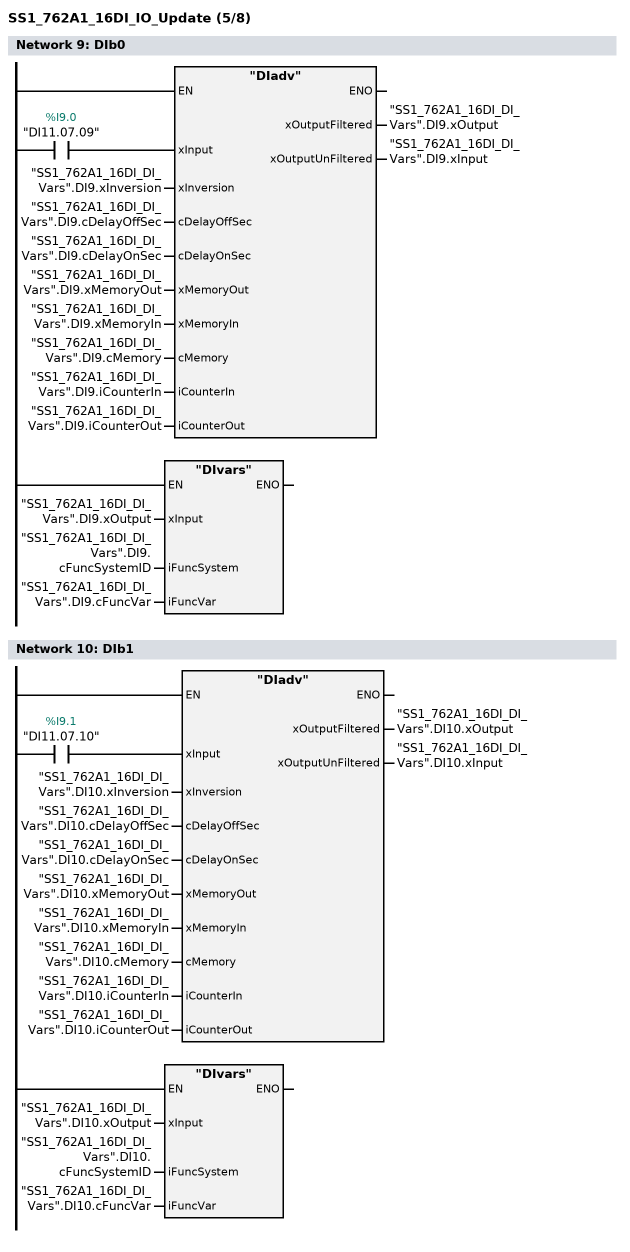
   RUNG wire#powerrail
      "DIadv"(xInput := wire#w1, xInversion := "SS1_762A1_16DI_DI_Vars".DI9.xInversion, cDelayOffSec := "SS1_762A1_16DI_DI_Vars".DI9.cDelayOffSec, cDelayOnSec := "SS1_762A1_16DI_DI_Vars".DI9.cDelayOnSec, xMemoryOut := "SS1_762A1_16DI_DI_Vars".DI9.xMemoryOut, xMemoryIn := "SS1_762A1_16DI_DI_Vars".DI9.xMemoryIn, cMemory := "SS1_762A1_16DI_DI_Vars".DI9.cMemory, iCounterIn := "SS1_762A1_16DI_DI_Vars".DI9.iCounterIn, iCounterOut := "SS1_762A1_16DI_DI_Vars".DI9.iCounterOut, xOutputFiltered => "SS1_762A1_16DI_DI_Vars".DI9.xOutput, xOutputUnFiltered => "SS1_762A1_16DI_DI_Vars".DI9.xInput)
   END_RUNG
   RUNG wire#powerrail
      Contact( "DI11.07.09" )
   END_RUNG wire#w1
   RUNG wire#powerrail
      "DIvars"(xInput := "SS1_762A1_16DI_DI_Vars".DI9.xOutput, iFuncSystem := "SS1_762A1_16DI_DI_Vars".DI9.cFuncSystemID, iFuncVar := "SS1_762A1_16DI_DI_Vars".DI9.cFuncVar)
   END_RUNG
   // the same network as SCL:
   "DIadv"(xInput := "DI11.07.09",
           xInversion := "SS1_762A1_16DI_DI_Vars".DI9.xInversion,
           cDelayOffSec := "SS1_762A1_16DI_DI_Vars".DI9.cDelayOffSec,
           cDelayOnSec := "SS1_762A1_16DI_DI_Vars".DI9.cDelayOnSec,
           xMemoryOut := "SS1_762A1_16DI_DI_Vars".DI9.xMemoryOut,
           xMemoryIn := "SS1_762A1_16DI_DI_Vars".DI9.xMemoryIn,
           cMemory := "SS1_762A1_16DI_DI_Vars".DI9.cMemory,
           iCounterIn := "SS1_762A1_16DI_DI_Vars".DI9.iCounterIn,
           iCounterOut := "SS1_762A1_16DI_DI_Vars".DI9.iCounterOut,
           xOutputFiltered => "SS1_762A1_16DI_DI_Vars".DI9.xOutput,
           xOutputUnFiltered => "SS1_762A1_16DI_DI_Vars".DI9.xInput);
   "DIvars"(xInput := "SS1_762A1_16DI_DI_Vars".DI9.xOutput,
            iFuncSystem := "SS1_762A1_16DI_DI_Vars".DI9.cFuncSystemID,
            iFuncVar := "SS1_762A1_16DI_DI_Vars".DI9.cFuncVar);
END_REGION

REGION Network 10: DIb1
   RUNG wire#powerrail
      "DIadv"(xInput := wire#w1, xInversion := "SS1_762A1_16DI_DI_Vars".DI10.xInversion, cDelayOffSec := "SS1_762A1_16DI_DI_Vars".DI10.cDelayOffSec, cDelayOnSec := "SS1_762A1_16DI_DI_Vars".DI10.cDelayOnSec, xMemoryOut := "SS1_762A1_16DI_DI_Vars".DI10.xMemoryOut, xMemoryIn := "SS1_762A1_16DI_DI_Vars".DI10.xMemoryIn, cMemory := "SS1_762A1_16DI_DI_Vars".DI10.cMemory, iCounterIn := "SS1_762A1_16DI_DI_Vars".DI10.iCounterIn, iCounterOut := "SS1_762A1_16DI_DI_Vars".DI10.iCounterOut, xOutputFiltered => "SS1_762A1_16DI_DI_Vars".DI10.xOutput, xOutputUnFiltered => "SS1_762A1_16DI_DI_Vars".DI10.xInput)
   END_RUNG
   RUNG wire#powerrail
      Contact( "DI11.07.10" )
   END_RUNG wire#w1
   RUNG wire#powerrail
      "DIvars"(xInput := "SS1_762A1_16DI_DI_Vars".DI10.xOutput, iFuncSystem := "SS1_762A1_16DI_DI_Vars".DI10.cFuncSystemID, iFuncVar := "SS1_762A1_16DI_DI_Vars".DI10.cFuncVar)
   END_RUNG
   // the same network as SCL:
   "DIadv"(xInput := "DI11.07.10",
           xInversion := "SS1_762A1_16DI_DI_Vars".DI10.xInversion,
           cDelayOffSec := "SS1_762A1_16DI_DI_Vars".DI10.cDelayOffSec,
           cDelayOnSec := "SS1_762A1_16DI_DI_Vars".DI10.cDelayOnSec,
           xMemoryOut := "SS1_762A1_16DI_DI_Vars".DI10.xMemoryOut,
           xMemoryIn := "SS1_762A1_16DI_DI_Vars".DI10.xMemoryIn,
           cMemory := "SS1_762A1_16DI_DI_Vars".DI10.cMemory,
           iCounterIn := "SS1_762A1_16DI_DI_Vars".DI10.iCounterIn,
           iCounterOut := "SS1_762A1_16DI_DI_Vars".DI10.iCounterOut,
           xOutputFiltered => "SS1_762A1_16DI_DI_Vars".DI10.xOutput,
           xOutputUnFiltered => "SS1_762A1_16DI_DI_Vars".DI10.xInput);
   "DIvars"(xInput := "SS1_762A1_16DI_DI_Vars".DI10.xOutput,
            iFuncSystem := "SS1_762A1_16DI_DI_Vars".DI10.cFuncSystemID,
            iFuncVar := "SS1_762A1_16DI_DI_Vars".DI10.cFuncVar);
END_REGION

REGION Network 11: DIb2
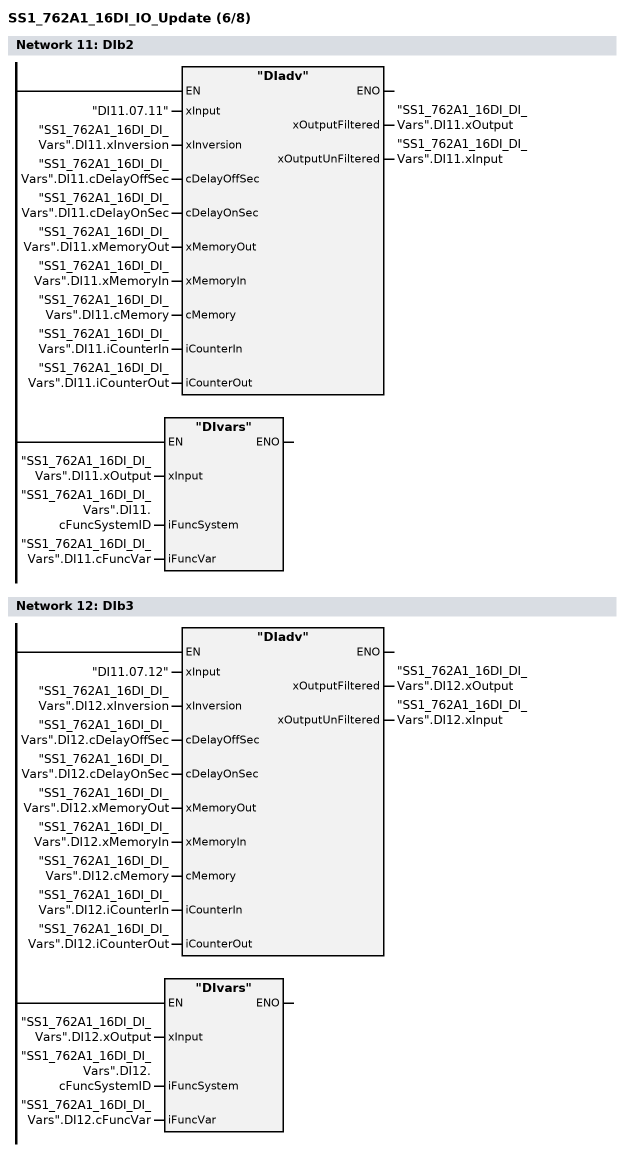
   RUNG wire#powerrail
      "DIadv"(xInput := "DI11.07.11", xInversion := "SS1_762A1_16DI_DI_Vars".DI11.xInversion, cDelayOffSec := "SS1_762A1_16DI_DI_Vars".DI11.cDelayOffSec, cDelayOnSec := "SS1_762A1_16DI_DI_Vars".DI11.cDelayOnSec, xMemoryOut := "SS1_762A1_16DI_DI_Vars".DI11.xMemoryOut, xMemoryIn := "SS1_762A1_16DI_DI_Vars".DI11.xMemoryIn, cMemory := "SS1_762A1_16DI_DI_Vars".DI11.cMemory, iCounterIn := "SS1_762A1_16DI_DI_Vars".DI11.iCounterIn, iCounterOut := "SS1_762A1_16DI_DI_Vars".DI11.iCounterOut, xOutputFiltered => "SS1_762A1_16DI_DI_Vars".DI11.xOutput, xOutputUnFiltered => "SS1_762A1_16DI_DI_Vars".DI11.xInput)
   END_RUNG
   RUNG wire#powerrail
      "DIvars"(xInput := "SS1_762A1_16DI_DI_Vars".DI11.xOutput, iFuncSystem := "SS1_762A1_16DI_DI_Vars".DI11.cFuncSystemID, iFuncVar := "SS1_762A1_16DI_DI_Vars".DI11.cFuncVar)
   END_RUNG
   // the same network as SCL:
   "DIadv"(xInput := "DI11.07.11",
           xInversion := "SS1_762A1_16DI_DI_Vars".DI11.xInversion,
           cDelayOffSec := "SS1_762A1_16DI_DI_Vars".DI11.cDelayOffSec,
           cDelayOnSec := "SS1_762A1_16DI_DI_Vars".DI11.cDelayOnSec,
           xMemoryOut := "SS1_762A1_16DI_DI_Vars".DI11.xMemoryOut,
           xMemoryIn := "SS1_762A1_16DI_DI_Vars".DI11.xMemoryIn,
           cMemory := "SS1_762A1_16DI_DI_Vars".DI11.cMemory,
           iCounterIn := "SS1_762A1_16DI_DI_Vars".DI11.iCounterIn,
           iCounterOut := "SS1_762A1_16DI_DI_Vars".DI11.iCounterOut,
           xOutputFiltered => "SS1_762A1_16DI_DI_Vars".DI11.xOutput,
           xOutputUnFiltered => "SS1_762A1_16DI_DI_Vars".DI11.xInput);
   "DIvars"(xInput := "SS1_762A1_16DI_DI_Vars".DI11.xOutput,
            iFuncSystem := "SS1_762A1_16DI_DI_Vars".DI11.cFuncSystemID,
            iFuncVar := "SS1_762A1_16DI_DI_Vars".DI11.cFuncVar);
END_REGION

REGION Network 12: DIb3
   RUNG wire#powerrail
      "DIadv"(xInput := "DI11.07.12", xInversion := "SS1_762A1_16DI_DI_Vars".DI12.xInversion, cDelayOffSec := "SS1_762A1_16DI_DI_Vars".DI12.cDelayOffSec, cDelayOnSec := "SS1_762A1_16DI_DI_Vars".DI12.cDelayOnSec, xMemoryOut := "SS1_762A1_16DI_DI_Vars".DI12.xMemoryOut, xMemoryIn := "SS1_762A1_16DI_DI_Vars".DI12.xMemoryIn, cMemory := "SS1_762A1_16DI_DI_Vars".DI12.cMemory, iCounterIn := "SS1_762A1_16DI_DI_Vars".DI12.iCounterIn, iCounterOut := "SS1_762A1_16DI_DI_Vars".DI12.iCounterOut, xOutputFiltered => "SS1_762A1_16DI_DI_Vars".DI12.xOutput, xOutputUnFiltered => "SS1_762A1_16DI_DI_Vars".DI12.xInput)
   END_RUNG
   RUNG wire#powerrail
      "DIvars"(xInput := "SS1_762A1_16DI_DI_Vars".DI12.xOutput, iFuncSystem := "SS1_762A1_16DI_DI_Vars".DI12.cFuncSystemID, iFuncVar := "SS1_762A1_16DI_DI_Vars".DI12.cFuncVar)
   END_RUNG
   // the same network as SCL:
   "DIadv"(xInput := "DI11.07.12",
           xInversion := "SS1_762A1_16DI_DI_Vars".DI12.xInversion,
           cDelayOffSec := "SS1_762A1_16DI_DI_Vars".DI12.cDelayOffSec,
           cDelayOnSec := "SS1_762A1_16DI_DI_Vars".DI12.cDelayOnSec,
           xMemoryOut := "SS1_762A1_16DI_DI_Vars".DI12.xMemoryOut,
           xMemoryIn := "SS1_762A1_16DI_DI_Vars".DI12.xMemoryIn,
           cMemory := "SS1_762A1_16DI_DI_Vars".DI12.cMemory,
           iCounterIn := "SS1_762A1_16DI_DI_Vars".DI12.iCounterIn,
           iCounterOut := "SS1_762A1_16DI_DI_Vars".DI12.iCounterOut,
           xOutputFiltered => "SS1_762A1_16DI_DI_Vars".DI12.xOutput,
           xOutputUnFiltered => "SS1_762A1_16DI_DI_Vars".DI12.xInput);
   "DIvars"(xInput := "SS1_762A1_16DI_DI_Vars".DI12.xOutput,
            iFuncSystem := "SS1_762A1_16DI_DI_Vars".DI12.cFuncSystemID,
            iFuncVar := "SS1_762A1_16DI_DI_Vars".DI12.cFuncVar);
END_REGION

REGION Network 13: DIb4
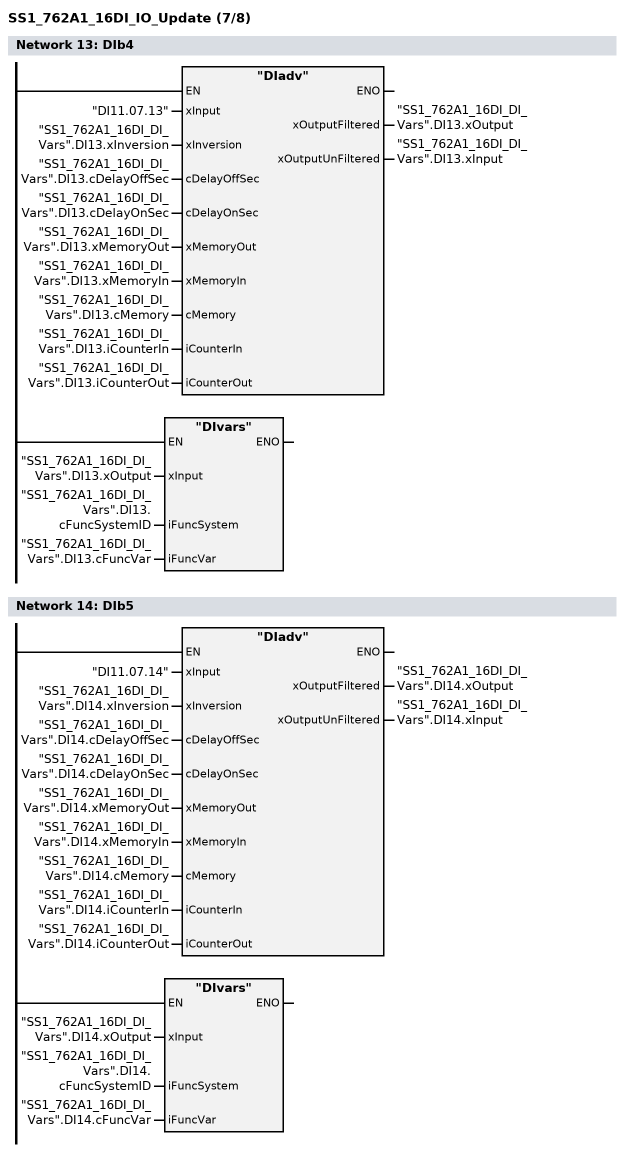
   RUNG wire#powerrail
      "DIadv"(xInput := "DI11.07.13", xInversion := "SS1_762A1_16DI_DI_Vars".DI13.xInversion, cDelayOffSec := "SS1_762A1_16DI_DI_Vars".DI13.cDelayOffSec, cDelayOnSec := "SS1_762A1_16DI_DI_Vars".DI13.cDelayOnSec, xMemoryOut := "SS1_762A1_16DI_DI_Vars".DI13.xMemoryOut, xMemoryIn := "SS1_762A1_16DI_DI_Vars".DI13.xMemoryIn, cMemory := "SS1_762A1_16DI_DI_Vars".DI13.cMemory, iCounterIn := "SS1_762A1_16DI_DI_Vars".DI13.iCounterIn, iCounterOut := "SS1_762A1_16DI_DI_Vars".DI13.iCounterOut, xOutputFiltered => "SS1_762A1_16DI_DI_Vars".DI13.xOutput, xOutputUnFiltered => "SS1_762A1_16DI_DI_Vars".DI13.xInput)
   END_RUNG
   RUNG wire#powerrail
      "DIvars"(xInput := "SS1_762A1_16DI_DI_Vars".DI13.xOutput, iFuncSystem := "SS1_762A1_16DI_DI_Vars".DI13.cFuncSystemID, iFuncVar := "SS1_762A1_16DI_DI_Vars".DI13.cFuncVar)
   END_RUNG
   // the same network as SCL:
   "DIadv"(xInput := "DI11.07.13",
           xInversion := "SS1_762A1_16DI_DI_Vars".DI13.xInversion,
           cDelayOffSec := "SS1_762A1_16DI_DI_Vars".DI13.cDelayOffSec,
           cDelayOnSec := "SS1_762A1_16DI_DI_Vars".DI13.cDelayOnSec,
           xMemoryOut := "SS1_762A1_16DI_DI_Vars".DI13.xMemoryOut,
           xMemoryIn := "SS1_762A1_16DI_DI_Vars".DI13.xMemoryIn,
           cMemory := "SS1_762A1_16DI_DI_Vars".DI13.cMemory,
           iCounterIn := "SS1_762A1_16DI_DI_Vars".DI13.iCounterIn,
           iCounterOut := "SS1_762A1_16DI_DI_Vars".DI13.iCounterOut,
           xOutputFiltered => "SS1_762A1_16DI_DI_Vars".DI13.xOutput,
           xOutputUnFiltered => "SS1_762A1_16DI_DI_Vars".DI13.xInput);
   "DIvars"(xInput := "SS1_762A1_16DI_DI_Vars".DI13.xOutput,
            iFuncSystem := "SS1_762A1_16DI_DI_Vars".DI13.cFuncSystemID,
            iFuncVar := "SS1_762A1_16DI_DI_Vars".DI13.cFuncVar);
END_REGION

REGION Network 14: DIb5
   RUNG wire#powerrail
      "DIadv"(xInput := "DI11.07.14", xInversion := "SS1_762A1_16DI_DI_Vars".DI14.xInversion, cDelayOffSec := "SS1_762A1_16DI_DI_Vars".DI14.cDelayOffSec, cDelayOnSec := "SS1_762A1_16DI_DI_Vars".DI14.cDelayOnSec, xMemoryOut := "SS1_762A1_16DI_DI_Vars".DI14.xMemoryOut, xMemoryIn := "SS1_762A1_16DI_DI_Vars".DI14.xMemoryIn, cMemory := "SS1_762A1_16DI_DI_Vars".DI14.cMemory, iCounterIn := "SS1_762A1_16DI_DI_Vars".DI14.iCounterIn, iCounterOut := "SS1_762A1_16DI_DI_Vars".DI14.iCounterOut, xOutputFiltered => "SS1_762A1_16DI_DI_Vars".DI14.xOutput, xOutputUnFiltered => "SS1_762A1_16DI_DI_Vars".DI14.xInput)
   END_RUNG
   RUNG wire#powerrail
      "DIvars"(xInput := "SS1_762A1_16DI_DI_Vars".DI14.xOutput, iFuncSystem := "SS1_762A1_16DI_DI_Vars".DI14.cFuncSystemID, iFuncVar := "SS1_762A1_16DI_DI_Vars".DI14.cFuncVar)
   END_RUNG
   // the same network as SCL:
   "DIadv"(xInput := "DI11.07.14",
           xInversion := "SS1_762A1_16DI_DI_Vars".DI14.xInversion,
           cDelayOffSec := "SS1_762A1_16DI_DI_Vars".DI14.cDelayOffSec,
           cDelayOnSec := "SS1_762A1_16DI_DI_Vars".DI14.cDelayOnSec,
           xMemoryOut := "SS1_762A1_16DI_DI_Vars".DI14.xMemoryOut,
           xMemoryIn := "SS1_762A1_16DI_DI_Vars".DI14.xMemoryIn,
           cMemory := "SS1_762A1_16DI_DI_Vars".DI14.cMemory,
           iCounterIn := "SS1_762A1_16DI_DI_Vars".DI14.iCounterIn,
           iCounterOut := "SS1_762A1_16DI_DI_Vars".DI14.iCounterOut,
           xOutputFiltered => "SS1_762A1_16DI_DI_Vars".DI14.xOutput,
           xOutputUnFiltered => "SS1_762A1_16DI_DI_Vars".DI14.xInput);
   "DIvars"(xInput := "SS1_762A1_16DI_DI_Vars".DI14.xOutput,
            iFuncSystem := "SS1_762A1_16DI_DI_Vars".DI14.cFuncSystemID,
            iFuncVar := "SS1_762A1_16DI_DI_Vars".DI14.cFuncVar);
END_REGION

REGION Network 15: DIb6
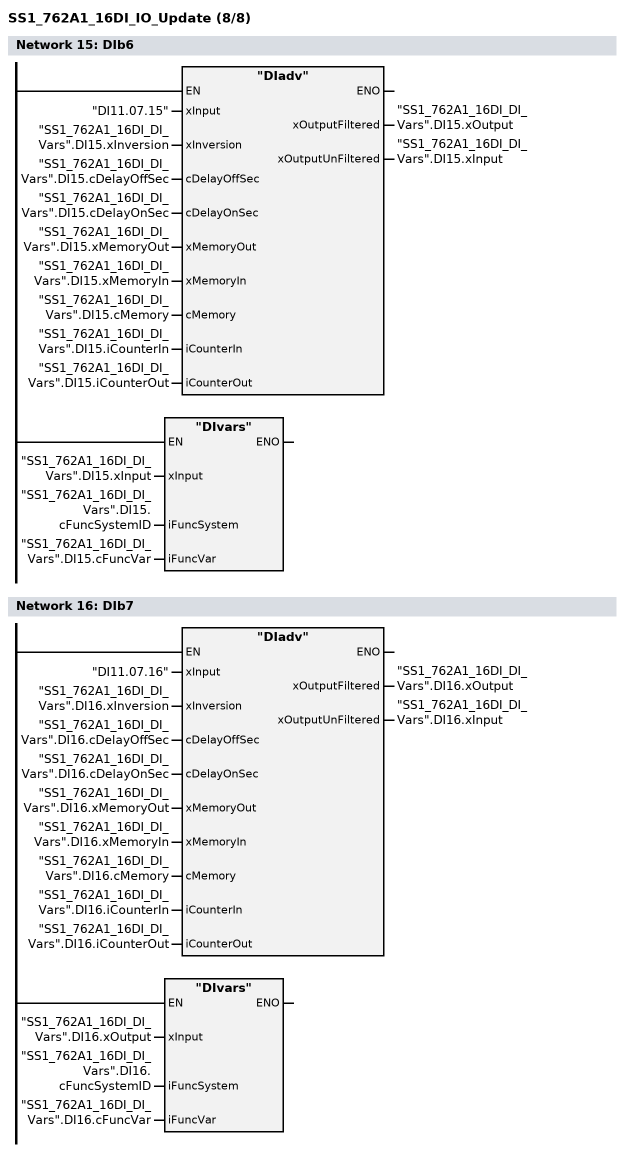
   RUNG wire#powerrail
      "DIadv"(xInput := "DI11.07.15", xInversion := "SS1_762A1_16DI_DI_Vars".DI15.xInversion, cDelayOffSec := "SS1_762A1_16DI_DI_Vars".DI15.cDelayOffSec, cDelayOnSec := "SS1_762A1_16DI_DI_Vars".DI15.cDelayOnSec, xMemoryOut := "SS1_762A1_16DI_DI_Vars".DI15.xMemoryOut, xMemoryIn := "SS1_762A1_16DI_DI_Vars".DI15.xMemoryIn, cMemory := "SS1_762A1_16DI_DI_Vars".DI15.cMemory, iCounterIn := "SS1_762A1_16DI_DI_Vars".DI15.iCounterIn, iCounterOut := "SS1_762A1_16DI_DI_Vars".DI15.iCounterOut, xOutputFiltered => "SS1_762A1_16DI_DI_Vars".DI15.xOutput, xOutputUnFiltered => "SS1_762A1_16DI_DI_Vars".DI15.xInput)
   END_RUNG
   RUNG wire#powerrail
      "DIvars"(xInput := "SS1_762A1_16DI_DI_Vars".DI15.xInput, iFuncSystem := "SS1_762A1_16DI_DI_Vars".DI15.cFuncSystemID, iFuncVar := "SS1_762A1_16DI_DI_Vars".DI15.cFuncVar)
   END_RUNG
   // the same network as SCL:
   "DIadv"(xInput := "DI11.07.15",
           xInversion := "SS1_762A1_16DI_DI_Vars".DI15.xInversion,
           cDelayOffSec := "SS1_762A1_16DI_DI_Vars".DI15.cDelayOffSec,
           cDelayOnSec := "SS1_762A1_16DI_DI_Vars".DI15.cDelayOnSec,
           xMemoryOut := "SS1_762A1_16DI_DI_Vars".DI15.xMemoryOut,
           xMemoryIn := "SS1_762A1_16DI_DI_Vars".DI15.xMemoryIn,
           cMemory := "SS1_762A1_16DI_DI_Vars".DI15.cMemory,
           iCounterIn := "SS1_762A1_16DI_DI_Vars".DI15.iCounterIn,
           iCounterOut := "SS1_762A1_16DI_DI_Vars".DI15.iCounterOut,
           xOutputFiltered => "SS1_762A1_16DI_DI_Vars".DI15.xOutput,
           xOutputUnFiltered => "SS1_762A1_16DI_DI_Vars".DI15.xInput);
   "DIvars"(xInput := "SS1_762A1_16DI_DI_Vars".DI15.xInput,
            iFuncSystem := "SS1_762A1_16DI_DI_Vars".DI15.cFuncSystemID,
            iFuncVar := "SS1_762A1_16DI_DI_Vars".DI15.cFuncVar);
END_REGION

REGION Network 16: DIb7
   RUNG wire#powerrail
      "DIadv"(xInput := "DI11.07.16", xInversion := "SS1_762A1_16DI_DI_Vars".DI16.xInversion, cDelayOffSec := "SS1_762A1_16DI_DI_Vars".DI16.cDelayOffSec, cDelayOnSec := "SS1_762A1_16DI_DI_Vars".DI16.cDelayOnSec, xMemoryOut := "SS1_762A1_16DI_DI_Vars".DI16.xMemoryOut, xMemoryIn := "SS1_762A1_16DI_DI_Vars".DI16.xMemoryIn, cMemory := "SS1_762A1_16DI_DI_Vars".DI16.cMemory, iCounterIn := "SS1_762A1_16DI_DI_Vars".DI16.iCounterIn, iCounterOut := "SS1_762A1_16DI_DI_Vars".DI16.iCounterOut, xOutputFiltered => "SS1_762A1_16DI_DI_Vars".DI16.xOutput, xOutputUnFiltered => "SS1_762A1_16DI_DI_Vars".DI16.xInput)
   END_RUNG
   RUNG wire#powerrail
      "DIvars"(xInput := "SS1_762A1_16DI_DI_Vars".DI16.xOutput, iFuncSystem := "SS1_762A1_16DI_DI_Vars".DI16.cFuncSystemID, iFuncVar := "SS1_762A1_16DI_DI_Vars".DI16.cFuncVar)
   END_RUNG
   // the same network as SCL:
   "DIadv"(xInput := "DI11.07.16",
           xInversion := "SS1_762A1_16DI_DI_Vars".DI16.xInversion,
           cDelayOffSec := "SS1_762A1_16DI_DI_Vars".DI16.cDelayOffSec,
           cDelayOnSec := "SS1_762A1_16DI_DI_Vars".DI16.cDelayOnSec,
           xMemoryOut := "SS1_762A1_16DI_DI_Vars".DI16.xMemoryOut,
           xMemoryIn := "SS1_762A1_16DI_DI_Vars".DI16.xMemoryIn,
           cMemory := "SS1_762A1_16DI_DI_Vars".DI16.cMemory,
           iCounterIn := "SS1_762A1_16DI_DI_Vars".DI16.iCounterIn,
           iCounterOut := "SS1_762A1_16DI_DI_Vars".DI16.iCounterOut,
           xOutputFiltered => "SS1_762A1_16DI_DI_Vars".DI16.xOutput,
           xOutputUnFiltered => "SS1_762A1_16DI_DI_Vars".DI16.xInput);
   "DIvars"(xInput := "SS1_762A1_16DI_DI_Vars".DI16.xOutput,
            iFuncSystem := "SS1_762A1_16DI_DI_Vars".DI16.cFuncSystemID,
            iFuncVar := "SS1_762A1_16DI_DI_Vars".DI16.cFuncVar);
END_REGION
END_FUNCTION

FUNCTION "SS1_770A1_16DO_IO_Update" : Void   // FC11070, LAD
{ S7_Optimized_Access := 'TRUE' }
VERSION : 0.1
// stored: AutoNumber false, IsIECCheckEnabled false, SetENOAutomatically false, UDAEnableTagReadback false
BEGIN

REGION Network 1: DQa0
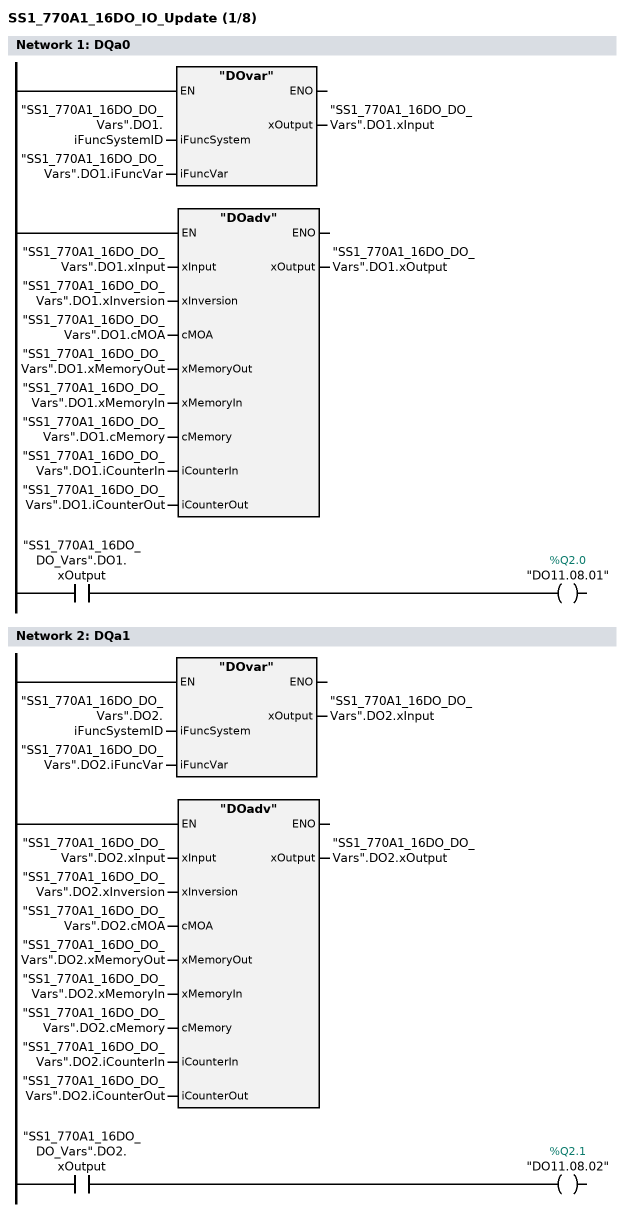
   RUNG wire#powerrail
      "DOvar"(iFuncSystem := "SS1_770A1_16DO_DO_Vars".DO1.iFuncSystemID, iFuncVar := "SS1_770A1_16DO_DO_Vars".DO1.iFuncVar, xOutput => "SS1_770A1_16DO_DO_Vars".DO1.xInput)
   END_RUNG
   RUNG wire#powerrail
      "DOadv"(xInput := "SS1_770A1_16DO_DO_Vars".DO1.xInput, xInversion := "SS1_770A1_16DO_DO_Vars".DO1.xInversion, cMOA := "SS1_770A1_16DO_DO_Vars".DO1.cMOA, xMemoryOut := "SS1_770A1_16DO_DO_Vars".DO1.xMemoryOut, xMemoryIn := "SS1_770A1_16DO_DO_Vars".DO1.xMemoryIn, cMemory := "SS1_770A1_16DO_DO_Vars".DO1.cMemory, iCounterIn := "SS1_770A1_16DO_DO_Vars".DO1.iCounterIn, iCounterOut := "SS1_770A1_16DO_DO_Vars".DO1.iCounterOut, xOutput => "SS1_770A1_16DO_DO_Vars".DO1.xOutput)
   END_RUNG
   RUNG wire#powerrail
      Contact( "SS1_770A1_16DO_DO_Vars".DO1.xOutput )
      Coil( "DO11.08.01" )
   END_RUNG
   // the same network as SCL:
   "DOvar"(iFuncSystem := "SS1_770A1_16DO_DO_Vars".DO1.iFuncSystemID,
           iFuncVar := "SS1_770A1_16DO_DO_Vars".DO1.iFuncVar,
           xOutput => "SS1_770A1_16DO_DO_Vars".DO1.xInput);
   "DOadv"(xInput := "SS1_770A1_16DO_DO_Vars".DO1.xInput,
           xInversion := "SS1_770A1_16DO_DO_Vars".DO1.xInversion,
           cMOA := "SS1_770A1_16DO_DO_Vars".DO1.cMOA,
           xMemoryOut := "SS1_770A1_16DO_DO_Vars".DO1.xMemoryOut,
           xMemoryIn := "SS1_770A1_16DO_DO_Vars".DO1.xMemoryIn,
           cMemory := "SS1_770A1_16DO_DO_Vars".DO1.cMemory,
           iCounterIn := "SS1_770A1_16DO_DO_Vars".DO1.iCounterIn,
           iCounterOut := "SS1_770A1_16DO_DO_Vars".DO1.iCounterOut,
           xOutput => "SS1_770A1_16DO_DO_Vars".DO1.xOutput);
   "DO11.08.01" := "SS1_770A1_16DO_DO_Vars".DO1.xOutput;
END_REGION

REGION Network 2: DQa1
   RUNG wire#powerrail
      "DOvar"(iFuncSystem := "SS1_770A1_16DO_DO_Vars".DO2.iFuncSystemID, iFuncVar := "SS1_770A1_16DO_DO_Vars".DO2.iFuncVar, xOutput => "SS1_770A1_16DO_DO_Vars".DO2.xInput)
   END_RUNG
   RUNG wire#powerrail
      "DOadv"(xInput := "SS1_770A1_16DO_DO_Vars".DO2.xInput, xInversion := "SS1_770A1_16DO_DO_Vars".DO2.xInversion, cMOA := "SS1_770A1_16DO_DO_Vars".DO2.cMOA, xMemoryOut := "SS1_770A1_16DO_DO_Vars".DO2.xMemoryOut, xMemoryIn := "SS1_770A1_16DO_DO_Vars".DO2.xMemoryIn, cMemory := "SS1_770A1_16DO_DO_Vars".DO2.cMemory, iCounterIn := "SS1_770A1_16DO_DO_Vars".DO2.iCounterIn, iCounterOut := "SS1_770A1_16DO_DO_Vars".DO2.iCounterOut, xOutput => "SS1_770A1_16DO_DO_Vars".DO2.xOutput)
   END_RUNG
   RUNG wire#powerrail
      Contact( "SS1_770A1_16DO_DO_Vars".DO2.xOutput )
      Coil( "DO11.08.02" )
   END_RUNG
   // the same network as SCL:
   "DOvar"(iFuncSystem := "SS1_770A1_16DO_DO_Vars".DO2.iFuncSystemID,
           iFuncVar := "SS1_770A1_16DO_DO_Vars".DO2.iFuncVar,
           xOutput => "SS1_770A1_16DO_DO_Vars".DO2.xInput);
   "DOadv"(xInput := "SS1_770A1_16DO_DO_Vars".DO2.xInput,
           xInversion := "SS1_770A1_16DO_DO_Vars".DO2.xInversion,
           cMOA := "SS1_770A1_16DO_DO_Vars".DO2.cMOA,
           xMemoryOut := "SS1_770A1_16DO_DO_Vars".DO2.xMemoryOut,
           xMemoryIn := "SS1_770A1_16DO_DO_Vars".DO2.xMemoryIn,
           cMemory := "SS1_770A1_16DO_DO_Vars".DO2.cMemory,
           iCounterIn := "SS1_770A1_16DO_DO_Vars".DO2.iCounterIn,
           iCounterOut := "SS1_770A1_16DO_DO_Vars".DO2.iCounterOut,
           xOutput => "SS1_770A1_16DO_DO_Vars".DO2.xOutput);
   "DO11.08.02" := "SS1_770A1_16DO_DO_Vars".DO2.xOutput;
END_REGION

REGION Network 3: DQa2
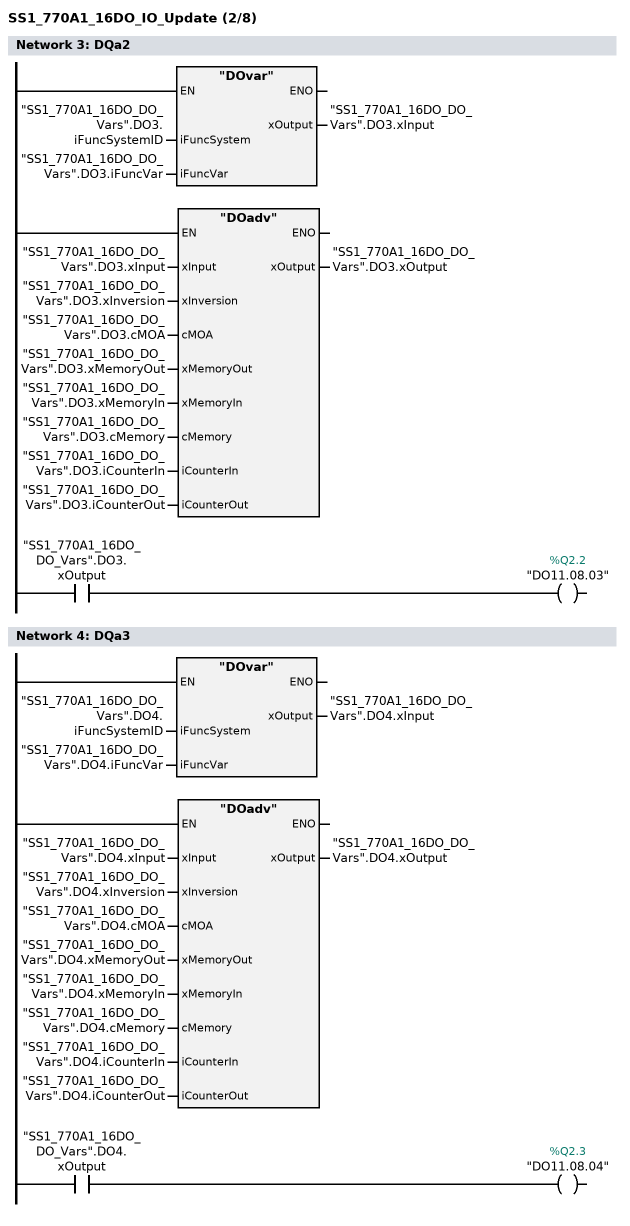
   RUNG wire#powerrail
      "DOvar"(iFuncSystem := "SS1_770A1_16DO_DO_Vars".DO3.iFuncSystemID, iFuncVar := "SS1_770A1_16DO_DO_Vars".DO3.iFuncVar, xOutput => "SS1_770A1_16DO_DO_Vars".DO3.xInput)
   END_RUNG
   RUNG wire#powerrail
      "DOadv"(xInput := "SS1_770A1_16DO_DO_Vars".DO3.xInput, xInversion := "SS1_770A1_16DO_DO_Vars".DO3.xInversion, cMOA := "SS1_770A1_16DO_DO_Vars".DO3.cMOA, xMemoryOut := "SS1_770A1_16DO_DO_Vars".DO3.xMemoryOut, xMemoryIn := "SS1_770A1_16DO_DO_Vars".DO3.xMemoryIn, cMemory := "SS1_770A1_16DO_DO_Vars".DO3.cMemory, iCounterIn := "SS1_770A1_16DO_DO_Vars".DO3.iCounterIn, iCounterOut := "SS1_770A1_16DO_DO_Vars".DO3.iCounterOut, xOutput => "SS1_770A1_16DO_DO_Vars".DO3.xOutput)
   END_RUNG
   RUNG wire#powerrail
      Contact( "SS1_770A1_16DO_DO_Vars".DO3.xOutput )
      Coil( "DO11.08.03" )
   END_RUNG
   // the same network as SCL:
   "DOvar"(iFuncSystem := "SS1_770A1_16DO_DO_Vars".DO3.iFuncSystemID,
           iFuncVar := "SS1_770A1_16DO_DO_Vars".DO3.iFuncVar,
           xOutput => "SS1_770A1_16DO_DO_Vars".DO3.xInput);
   "DOadv"(xInput := "SS1_770A1_16DO_DO_Vars".DO3.xInput,
           xInversion := "SS1_770A1_16DO_DO_Vars".DO3.xInversion,
           cMOA := "SS1_770A1_16DO_DO_Vars".DO3.cMOA,
           xMemoryOut := "SS1_770A1_16DO_DO_Vars".DO3.xMemoryOut,
           xMemoryIn := "SS1_770A1_16DO_DO_Vars".DO3.xMemoryIn,
           cMemory := "SS1_770A1_16DO_DO_Vars".DO3.cMemory,
           iCounterIn := "SS1_770A1_16DO_DO_Vars".DO3.iCounterIn,
           iCounterOut := "SS1_770A1_16DO_DO_Vars".DO3.iCounterOut,
           xOutput => "SS1_770A1_16DO_DO_Vars".DO3.xOutput);
   "DO11.08.03" := "SS1_770A1_16DO_DO_Vars".DO3.xOutput;
END_REGION

REGION Network 4: DQa3
   RUNG wire#powerrail
      "DOvar"(iFuncSystem := "SS1_770A1_16DO_DO_Vars".DO4.iFuncSystemID, iFuncVar := "SS1_770A1_16DO_DO_Vars".DO4.iFuncVar, xOutput => "SS1_770A1_16DO_DO_Vars".DO4.xInput)
   END_RUNG
   RUNG wire#powerrail
      "DOadv"(xInput := "SS1_770A1_16DO_DO_Vars".DO4.xInput, xInversion := "SS1_770A1_16DO_DO_Vars".DO4.xInversion, cMOA := "SS1_770A1_16DO_DO_Vars".DO4.cMOA, xMemoryOut := "SS1_770A1_16DO_DO_Vars".DO4.xMemoryOut, xMemoryIn := "SS1_770A1_16DO_DO_Vars".DO4.xMemoryIn, cMemory := "SS1_770A1_16DO_DO_Vars".DO4.cMemory, iCounterIn := "SS1_770A1_16DO_DO_Vars".DO4.iCounterIn, iCounterOut := "SS1_770A1_16DO_DO_Vars".DO4.iCounterOut, xOutput => "SS1_770A1_16DO_DO_Vars".DO4.xOutput)
   END_RUNG
   RUNG wire#powerrail
      Contact( "SS1_770A1_16DO_DO_Vars".DO4.xOutput )
      Coil( "DO11.08.04" )
   END_RUNG
   // the same network as SCL:
   "DOvar"(iFuncSystem := "SS1_770A1_16DO_DO_Vars".DO4.iFuncSystemID,
           iFuncVar := "SS1_770A1_16DO_DO_Vars".DO4.iFuncVar,
           xOutput => "SS1_770A1_16DO_DO_Vars".DO4.xInput);
   "DOadv"(xInput := "SS1_770A1_16DO_DO_Vars".DO4.xInput,
           xInversion := "SS1_770A1_16DO_DO_Vars".DO4.xInversion,
           cMOA := "SS1_770A1_16DO_DO_Vars".DO4.cMOA,
           xMemoryOut := "SS1_770A1_16DO_DO_Vars".DO4.xMemoryOut,
           xMemoryIn := "SS1_770A1_16DO_DO_Vars".DO4.xMemoryIn,
           cMemory := "SS1_770A1_16DO_DO_Vars".DO4.cMemory,
           iCounterIn := "SS1_770A1_16DO_DO_Vars".DO4.iCounterIn,
           iCounterOut := "SS1_770A1_16DO_DO_Vars".DO4.iCounterOut,
           xOutput => "SS1_770A1_16DO_DO_Vars".DO4.xOutput);
   "DO11.08.04" := "SS1_770A1_16DO_DO_Vars".DO4.xOutput;
END_REGION

REGION Network 5: DQa4
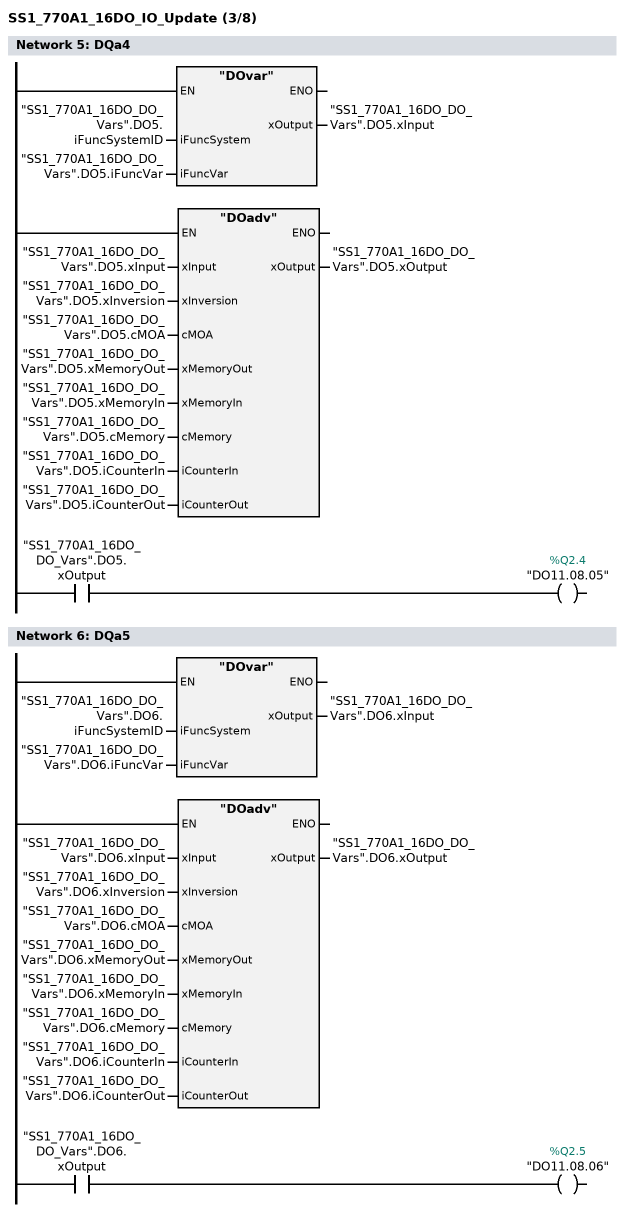
   RUNG wire#powerrail
      "DOvar"(iFuncSystem := "SS1_770A1_16DO_DO_Vars".DO5.iFuncSystemID, iFuncVar := "SS1_770A1_16DO_DO_Vars".DO5.iFuncVar, xOutput => "SS1_770A1_16DO_DO_Vars".DO5.xInput)
   END_RUNG
   RUNG wire#powerrail
      "DOadv"(xInput := "SS1_770A1_16DO_DO_Vars".DO5.xInput, xInversion := "SS1_770A1_16DO_DO_Vars".DO5.xInversion, cMOA := "SS1_770A1_16DO_DO_Vars".DO5.cMOA, xMemoryOut := "SS1_770A1_16DO_DO_Vars".DO5.xMemoryOut, xMemoryIn := "SS1_770A1_16DO_DO_Vars".DO5.xMemoryIn, cMemory := "SS1_770A1_16DO_DO_Vars".DO5.cMemory, iCounterIn := "SS1_770A1_16DO_DO_Vars".DO5.iCounterIn, iCounterOut := "SS1_770A1_16DO_DO_Vars".DO5.iCounterOut, xOutput => "SS1_770A1_16DO_DO_Vars".DO5.xOutput)
   END_RUNG
   RUNG wire#powerrail
      Contact( "SS1_770A1_16DO_DO_Vars".DO5.xOutput )
      Coil( "DO11.08.05" )
   END_RUNG
   // the same network as SCL:
   "DOvar"(iFuncSystem := "SS1_770A1_16DO_DO_Vars".DO5.iFuncSystemID,
           iFuncVar := "SS1_770A1_16DO_DO_Vars".DO5.iFuncVar,
           xOutput => "SS1_770A1_16DO_DO_Vars".DO5.xInput);
   "DOadv"(xInput := "SS1_770A1_16DO_DO_Vars".DO5.xInput,
           xInversion := "SS1_770A1_16DO_DO_Vars".DO5.xInversion,
           cMOA := "SS1_770A1_16DO_DO_Vars".DO5.cMOA,
           xMemoryOut := "SS1_770A1_16DO_DO_Vars".DO5.xMemoryOut,
           xMemoryIn := "SS1_770A1_16DO_DO_Vars".DO5.xMemoryIn,
           cMemory := "SS1_770A1_16DO_DO_Vars".DO5.cMemory,
           iCounterIn := "SS1_770A1_16DO_DO_Vars".DO5.iCounterIn,
           iCounterOut := "SS1_770A1_16DO_DO_Vars".DO5.iCounterOut,
           xOutput => "SS1_770A1_16DO_DO_Vars".DO5.xOutput);
   "DO11.08.05" := "SS1_770A1_16DO_DO_Vars".DO5.xOutput;
END_REGION

REGION Network 6: DQa5
   RUNG wire#powerrail
      "DOvar"(iFuncSystem := "SS1_770A1_16DO_DO_Vars".DO6.iFuncSystemID, iFuncVar := "SS1_770A1_16DO_DO_Vars".DO6.iFuncVar, xOutput => "SS1_770A1_16DO_DO_Vars".DO6.xInput)
   END_RUNG
   RUNG wire#powerrail
      "DOadv"(xInput := "SS1_770A1_16DO_DO_Vars".DO6.xInput, xInversion := "SS1_770A1_16DO_DO_Vars".DO6.xInversion, cMOA := "SS1_770A1_16DO_DO_Vars".DO6.cMOA, xMemoryOut := "SS1_770A1_16DO_DO_Vars".DO6.xMemoryOut, xMemoryIn := "SS1_770A1_16DO_DO_Vars".DO6.xMemoryIn, cMemory := "SS1_770A1_16DO_DO_Vars".DO6.cMemory, iCounterIn := "SS1_770A1_16DO_DO_Vars".DO6.iCounterIn, iCounterOut := "SS1_770A1_16DO_DO_Vars".DO6.iCounterOut, xOutput => "SS1_770A1_16DO_DO_Vars".DO6.xOutput)
   END_RUNG
   RUNG wire#powerrail
      Contact( "SS1_770A1_16DO_DO_Vars".DO6.xOutput )
      Coil( "DO11.08.06" )
   END_RUNG
   // the same network as SCL:
   "DOvar"(iFuncSystem := "SS1_770A1_16DO_DO_Vars".DO6.iFuncSystemID,
           iFuncVar := "SS1_770A1_16DO_DO_Vars".DO6.iFuncVar,
           xOutput => "SS1_770A1_16DO_DO_Vars".DO6.xInput);
   "DOadv"(xInput := "SS1_770A1_16DO_DO_Vars".DO6.xInput,
           xInversion := "SS1_770A1_16DO_DO_Vars".DO6.xInversion,
           cMOA := "SS1_770A1_16DO_DO_Vars".DO6.cMOA,
           xMemoryOut := "SS1_770A1_16DO_DO_Vars".DO6.xMemoryOut,
           xMemoryIn := "SS1_770A1_16DO_DO_Vars".DO6.xMemoryIn,
           cMemory := "SS1_770A1_16DO_DO_Vars".DO6.cMemory,
           iCounterIn := "SS1_770A1_16DO_DO_Vars".DO6.iCounterIn,
           iCounterOut := "SS1_770A1_16DO_DO_Vars".DO6.iCounterOut,
           xOutput => "SS1_770A1_16DO_DO_Vars".DO6.xOutput);
   "DO11.08.06" := "SS1_770A1_16DO_DO_Vars".DO6.xOutput;
END_REGION

REGION Network 7: DQa6
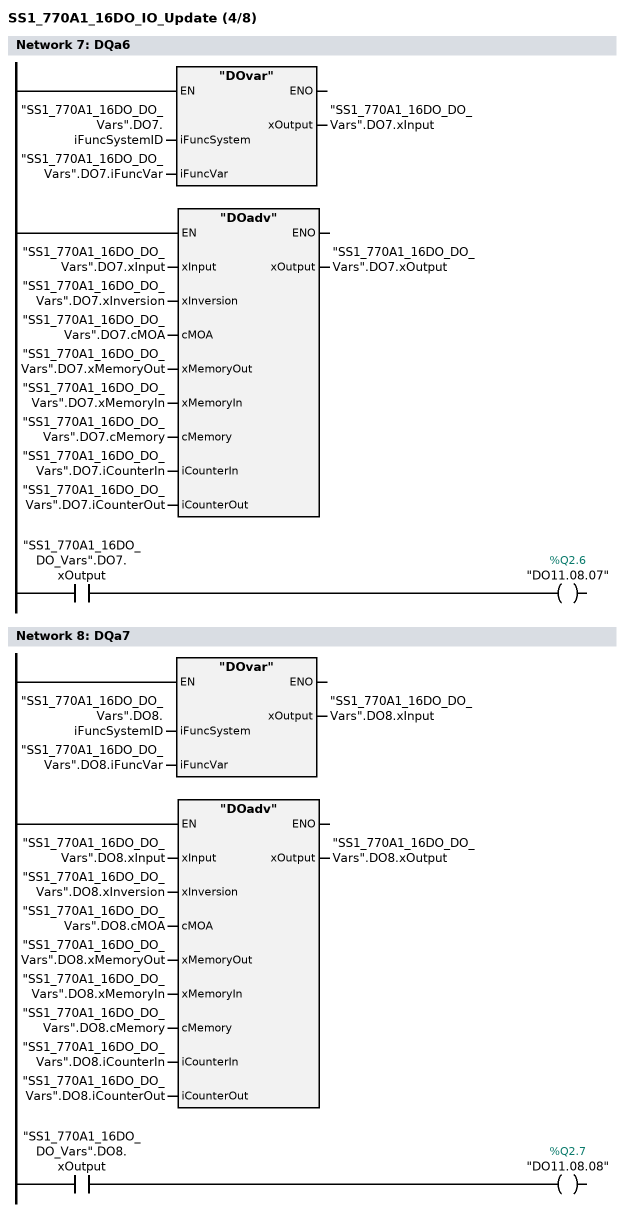
   RUNG wire#powerrail
      "DOvar"(iFuncSystem := "SS1_770A1_16DO_DO_Vars".DO7.iFuncSystemID, iFuncVar := "SS1_770A1_16DO_DO_Vars".DO7.iFuncVar, xOutput => "SS1_770A1_16DO_DO_Vars".DO7.xInput)
   END_RUNG
   RUNG wire#powerrail
      "DOadv"(xInput := "SS1_770A1_16DO_DO_Vars".DO7.xInput, xInversion := "SS1_770A1_16DO_DO_Vars".DO7.xInversion, cMOA := "SS1_770A1_16DO_DO_Vars".DO7.cMOA, xMemoryOut := "SS1_770A1_16DO_DO_Vars".DO7.xMemoryOut, xMemoryIn := "SS1_770A1_16DO_DO_Vars".DO7.xMemoryIn, cMemory := "SS1_770A1_16DO_DO_Vars".DO7.cMemory, iCounterIn := "SS1_770A1_16DO_DO_Vars".DO7.iCounterIn, iCounterOut := "SS1_770A1_16DO_DO_Vars".DO7.iCounterOut, xOutput => "SS1_770A1_16DO_DO_Vars".DO7.xOutput)
   END_RUNG
   RUNG wire#powerrail
      Contact( "SS1_770A1_16DO_DO_Vars".DO7.xOutput )
      Coil( "DO11.08.07" )
   END_RUNG
   // the same network as SCL:
   "DOvar"(iFuncSystem := "SS1_770A1_16DO_DO_Vars".DO7.iFuncSystemID,
           iFuncVar := "SS1_770A1_16DO_DO_Vars".DO7.iFuncVar,
           xOutput => "SS1_770A1_16DO_DO_Vars".DO7.xInput);
   "DOadv"(xInput := "SS1_770A1_16DO_DO_Vars".DO7.xInput,
           xInversion := "SS1_770A1_16DO_DO_Vars".DO7.xInversion,
           cMOA := "SS1_770A1_16DO_DO_Vars".DO7.cMOA,
           xMemoryOut := "SS1_770A1_16DO_DO_Vars".DO7.xMemoryOut,
           xMemoryIn := "SS1_770A1_16DO_DO_Vars".DO7.xMemoryIn,
           cMemory := "SS1_770A1_16DO_DO_Vars".DO7.cMemory,
           iCounterIn := "SS1_770A1_16DO_DO_Vars".DO7.iCounterIn,
           iCounterOut := "SS1_770A1_16DO_DO_Vars".DO7.iCounterOut,
           xOutput => "SS1_770A1_16DO_DO_Vars".DO7.xOutput);
   "DO11.08.07" := "SS1_770A1_16DO_DO_Vars".DO7.xOutput;
END_REGION

REGION Network 8: DQa7
   RUNG wire#powerrail
      "DOvar"(iFuncSystem := "SS1_770A1_16DO_DO_Vars".DO8.iFuncSystemID, iFuncVar := "SS1_770A1_16DO_DO_Vars".DO8.iFuncVar, xOutput => "SS1_770A1_16DO_DO_Vars".DO8.xInput)
   END_RUNG
   RUNG wire#powerrail
      "DOadv"(xInput := "SS1_770A1_16DO_DO_Vars".DO8.xInput, xInversion := "SS1_770A1_16DO_DO_Vars".DO8.xInversion, cMOA := "SS1_770A1_16DO_DO_Vars".DO8.cMOA, xMemoryOut := "SS1_770A1_16DO_DO_Vars".DO8.xMemoryOut, xMemoryIn := "SS1_770A1_16DO_DO_Vars".DO8.xMemoryIn, cMemory := "SS1_770A1_16DO_DO_Vars".DO8.cMemory, iCounterIn := "SS1_770A1_16DO_DO_Vars".DO8.iCounterIn, iCounterOut := "SS1_770A1_16DO_DO_Vars".DO8.iCounterOut, xOutput => "SS1_770A1_16DO_DO_Vars".DO8.xOutput)
   END_RUNG
   RUNG wire#powerrail
      Contact( "SS1_770A1_16DO_DO_Vars".DO8.xOutput )
      Coil( "DO11.08.08" )
   END_RUNG
   // the same network as SCL:
   "DOvar"(iFuncSystem := "SS1_770A1_16DO_DO_Vars".DO8.iFuncSystemID,
           iFuncVar := "SS1_770A1_16DO_DO_Vars".DO8.iFuncVar,
           xOutput => "SS1_770A1_16DO_DO_Vars".DO8.xInput);
   "DOadv"(xInput := "SS1_770A1_16DO_DO_Vars".DO8.xInput,
           xInversion := "SS1_770A1_16DO_DO_Vars".DO8.xInversion,
           cMOA := "SS1_770A1_16DO_DO_Vars".DO8.cMOA,
           xMemoryOut := "SS1_770A1_16DO_DO_Vars".DO8.xMemoryOut,
           xMemoryIn := "SS1_770A1_16DO_DO_Vars".DO8.xMemoryIn,
           cMemory := "SS1_770A1_16DO_DO_Vars".DO8.cMemory,
           iCounterIn := "SS1_770A1_16DO_DO_Vars".DO8.iCounterIn,
           iCounterOut := "SS1_770A1_16DO_DO_Vars".DO8.iCounterOut,
           xOutput => "SS1_770A1_16DO_DO_Vars".DO8.xOutput);
   "DO11.08.08" := "SS1_770A1_16DO_DO_Vars".DO8.xOutput;
END_REGION

REGION Network 9: DQb0
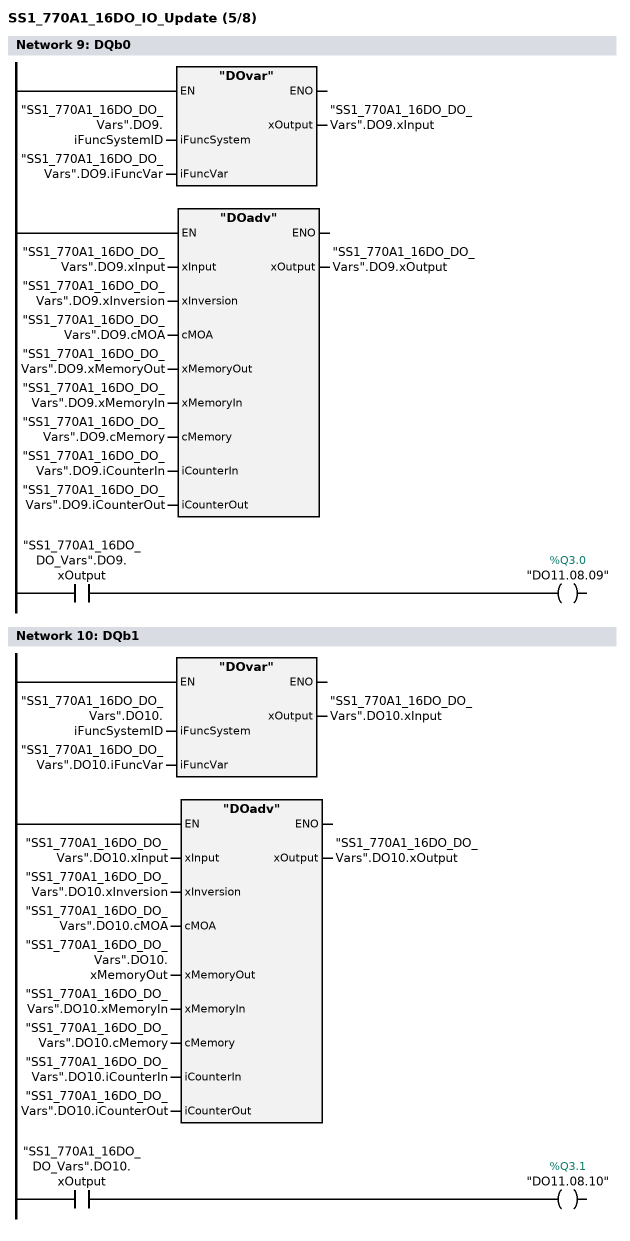
   RUNG wire#powerrail
      "DOvar"(iFuncSystem := "SS1_770A1_16DO_DO_Vars".DO9.iFuncSystemID, iFuncVar := "SS1_770A1_16DO_DO_Vars".DO9.iFuncVar, xOutput => "SS1_770A1_16DO_DO_Vars".DO9.xInput)
   END_RUNG
   RUNG wire#powerrail
      "DOadv"(xInput := "SS1_770A1_16DO_DO_Vars".DO9.xInput, xInversion := "SS1_770A1_16DO_DO_Vars".DO9.xInversion, cMOA := "SS1_770A1_16DO_DO_Vars".DO9.cMOA, xMemoryOut := "SS1_770A1_16DO_DO_Vars".DO9.xMemoryOut, xMemoryIn := "SS1_770A1_16DO_DO_Vars".DO9.xMemoryIn, cMemory := "SS1_770A1_16DO_DO_Vars".DO9.cMemory, iCounterIn := "SS1_770A1_16DO_DO_Vars".DO9.iCounterIn, iCounterOut := "SS1_770A1_16DO_DO_Vars".DO9.iCounterOut, xOutput => "SS1_770A1_16DO_DO_Vars".DO9.xOutput)
   END_RUNG
   RUNG wire#powerrail
      Contact( "SS1_770A1_16DO_DO_Vars".DO9.xOutput )
      Coil( "DO11.08.09" )
   END_RUNG
   // the same network as SCL:
   "DOvar"(iFuncSystem := "SS1_770A1_16DO_DO_Vars".DO9.iFuncSystemID,
           iFuncVar := "SS1_770A1_16DO_DO_Vars".DO9.iFuncVar,
           xOutput => "SS1_770A1_16DO_DO_Vars".DO9.xInput);
   "DOadv"(xInput := "SS1_770A1_16DO_DO_Vars".DO9.xInput,
           xInversion := "SS1_770A1_16DO_DO_Vars".DO9.xInversion,
           cMOA := "SS1_770A1_16DO_DO_Vars".DO9.cMOA,
           xMemoryOut := "SS1_770A1_16DO_DO_Vars".DO9.xMemoryOut,
           xMemoryIn := "SS1_770A1_16DO_DO_Vars".DO9.xMemoryIn,
           cMemory := "SS1_770A1_16DO_DO_Vars".DO9.cMemory,
           iCounterIn := "SS1_770A1_16DO_DO_Vars".DO9.iCounterIn,
           iCounterOut := "SS1_770A1_16DO_DO_Vars".DO9.iCounterOut,
           xOutput => "SS1_770A1_16DO_DO_Vars".DO9.xOutput);
   "DO11.08.09" := "SS1_770A1_16DO_DO_Vars".DO9.xOutput;
END_REGION

REGION Network 10: DQb1
   RUNG wire#powerrail
      "DOvar"(iFuncSystem := "SS1_770A1_16DO_DO_Vars".DO10.iFuncSystemID, iFuncVar := "SS1_770A1_16DO_DO_Vars".DO10.iFuncVar, xOutput => "SS1_770A1_16DO_DO_Vars".DO10.xInput)
   END_RUNG
   RUNG wire#powerrail
      "DOadv"(xInput := "SS1_770A1_16DO_DO_Vars".DO10.xInput, xInversion := "SS1_770A1_16DO_DO_Vars".DO10.xInversion, cMOA := "SS1_770A1_16DO_DO_Vars".DO10.cMOA, xMemoryOut := "SS1_770A1_16DO_DO_Vars".DO10.xMemoryOut, xMemoryIn := "SS1_770A1_16DO_DO_Vars".DO10.xMemoryIn, cMemory := "SS1_770A1_16DO_DO_Vars".DO10.cMemory, iCounterIn := "SS1_770A1_16DO_DO_Vars".DO10.iCounterIn, iCounterOut := "SS1_770A1_16DO_DO_Vars".DO10.iCounterOut, xOutput => "SS1_770A1_16DO_DO_Vars".DO10.xOutput)
   END_RUNG
   RUNG wire#powerrail
      Contact( "SS1_770A1_16DO_DO_Vars".DO10.xOutput )
      Coil( "DO11.08.10" )
   END_RUNG
   // the same network as SCL:
   "DOvar"(iFuncSystem := "SS1_770A1_16DO_DO_Vars".DO10.iFuncSystemID,
           iFuncVar := "SS1_770A1_16DO_DO_Vars".DO10.iFuncVar,
           xOutput => "SS1_770A1_16DO_DO_Vars".DO10.xInput);
   "DOadv"(xInput := "SS1_770A1_16DO_DO_Vars".DO10.xInput,
           xInversion := "SS1_770A1_16DO_DO_Vars".DO10.xInversion,
           cMOA := "SS1_770A1_16DO_DO_Vars".DO10.cMOA,
           xMemoryOut := "SS1_770A1_16DO_DO_Vars".DO10.xMemoryOut,
           xMemoryIn := "SS1_770A1_16DO_DO_Vars".DO10.xMemoryIn,
           cMemory := "SS1_770A1_16DO_DO_Vars".DO10.cMemory,
           iCounterIn := "SS1_770A1_16DO_DO_Vars".DO10.iCounterIn,
           iCounterOut := "SS1_770A1_16DO_DO_Vars".DO10.iCounterOut,
           xOutput => "SS1_770A1_16DO_DO_Vars".DO10.xOutput);
   "DO11.08.10" := "SS1_770A1_16DO_DO_Vars".DO10.xOutput;
END_REGION

REGION Network 11: DQb2
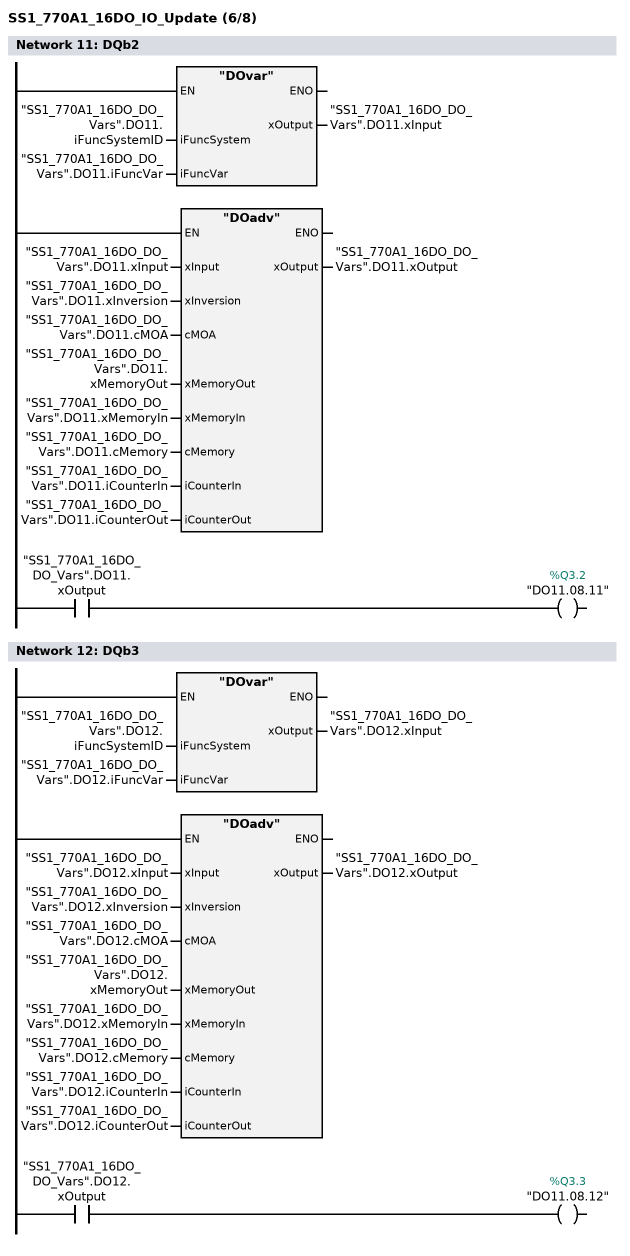
   RUNG wire#powerrail
      "DOvar"(iFuncSystem := "SS1_770A1_16DO_DO_Vars".DO11.iFuncSystemID, iFuncVar := "SS1_770A1_16DO_DO_Vars".DO11.iFuncVar, xOutput => "SS1_770A1_16DO_DO_Vars".DO11.xInput)
   END_RUNG
   RUNG wire#powerrail
      "DOadv"(xInput := "SS1_770A1_16DO_DO_Vars".DO11.xInput, xInversion := "SS1_770A1_16DO_DO_Vars".DO11.xInversion, cMOA := "SS1_770A1_16DO_DO_Vars".DO11.cMOA, xMemoryOut := "SS1_770A1_16DO_DO_Vars".DO11.xMemoryOut, xMemoryIn := "SS1_770A1_16DO_DO_Vars".DO11.xMemoryIn, cMemory := "SS1_770A1_16DO_DO_Vars".DO11.cMemory, iCounterIn := "SS1_770A1_16DO_DO_Vars".DO11.iCounterIn, iCounterOut := "SS1_770A1_16DO_DO_Vars".DO11.iCounterOut, xOutput => "SS1_770A1_16DO_DO_Vars".DO11.xOutput)
   END_RUNG
   RUNG wire#powerrail
      Contact( "SS1_770A1_16DO_DO_Vars".DO11.xOutput )
      Coil( "DO11.08.11" )
   END_RUNG
   // the same network as SCL:
   "DOvar"(iFuncSystem := "SS1_770A1_16DO_DO_Vars".DO11.iFuncSystemID,
           iFuncVar := "SS1_770A1_16DO_DO_Vars".DO11.iFuncVar,
           xOutput => "SS1_770A1_16DO_DO_Vars".DO11.xInput);
   "DOadv"(xInput := "SS1_770A1_16DO_DO_Vars".DO11.xInput,
           xInversion := "SS1_770A1_16DO_DO_Vars".DO11.xInversion,
           cMOA := "SS1_770A1_16DO_DO_Vars".DO11.cMOA,
           xMemoryOut := "SS1_770A1_16DO_DO_Vars".DO11.xMemoryOut,
           xMemoryIn := "SS1_770A1_16DO_DO_Vars".DO11.xMemoryIn,
           cMemory := "SS1_770A1_16DO_DO_Vars".DO11.cMemory,
           iCounterIn := "SS1_770A1_16DO_DO_Vars".DO11.iCounterIn,
           iCounterOut := "SS1_770A1_16DO_DO_Vars".DO11.iCounterOut,
           xOutput => "SS1_770A1_16DO_DO_Vars".DO11.xOutput);
   "DO11.08.11" := "SS1_770A1_16DO_DO_Vars".DO11.xOutput;
END_REGION

REGION Network 12: DQb3
   RUNG wire#powerrail
      "DOvar"(iFuncSystem := "SS1_770A1_16DO_DO_Vars".DO12.iFuncSystemID, iFuncVar := "SS1_770A1_16DO_DO_Vars".DO12.iFuncVar, xOutput => "SS1_770A1_16DO_DO_Vars".DO12.xInput)
   END_RUNG
   RUNG wire#powerrail
      "DOadv"(xInput := "SS1_770A1_16DO_DO_Vars".DO12.xInput, xInversion := "SS1_770A1_16DO_DO_Vars".DO12.xInversion, cMOA := "SS1_770A1_16DO_DO_Vars".DO12.cMOA, xMemoryOut := "SS1_770A1_16DO_DO_Vars".DO12.xMemoryOut, xMemoryIn := "SS1_770A1_16DO_DO_Vars".DO12.xMemoryIn, cMemory := "SS1_770A1_16DO_DO_Vars".DO12.cMemory, iCounterIn := "SS1_770A1_16DO_DO_Vars".DO12.iCounterIn, iCounterOut := "SS1_770A1_16DO_DO_Vars".DO12.iCounterOut, xOutput => "SS1_770A1_16DO_DO_Vars".DO12.xOutput)
   END_RUNG
   RUNG wire#powerrail
      Contact( "SS1_770A1_16DO_DO_Vars".DO12.xOutput )
      Coil( "DO11.08.12" )
   END_RUNG
   // the same network as SCL:
   "DOvar"(iFuncSystem := "SS1_770A1_16DO_DO_Vars".DO12.iFuncSystemID,
           iFuncVar := "SS1_770A1_16DO_DO_Vars".DO12.iFuncVar,
           xOutput => "SS1_770A1_16DO_DO_Vars".DO12.xInput);
   "DOadv"(xInput := "SS1_770A1_16DO_DO_Vars".DO12.xInput,
           xInversion := "SS1_770A1_16DO_DO_Vars".DO12.xInversion,
           cMOA := "SS1_770A1_16DO_DO_Vars".DO12.cMOA,
           xMemoryOut := "SS1_770A1_16DO_DO_Vars".DO12.xMemoryOut,
           xMemoryIn := "SS1_770A1_16DO_DO_Vars".DO12.xMemoryIn,
           cMemory := "SS1_770A1_16DO_DO_Vars".DO12.cMemory,
           iCounterIn := "SS1_770A1_16DO_DO_Vars".DO12.iCounterIn,
           iCounterOut := "SS1_770A1_16DO_DO_Vars".DO12.iCounterOut,
           xOutput => "SS1_770A1_16DO_DO_Vars".DO12.xOutput);
   "DO11.08.12" := "SS1_770A1_16DO_DO_Vars".DO12.xOutput;
END_REGION

REGION Network 13: DQb4
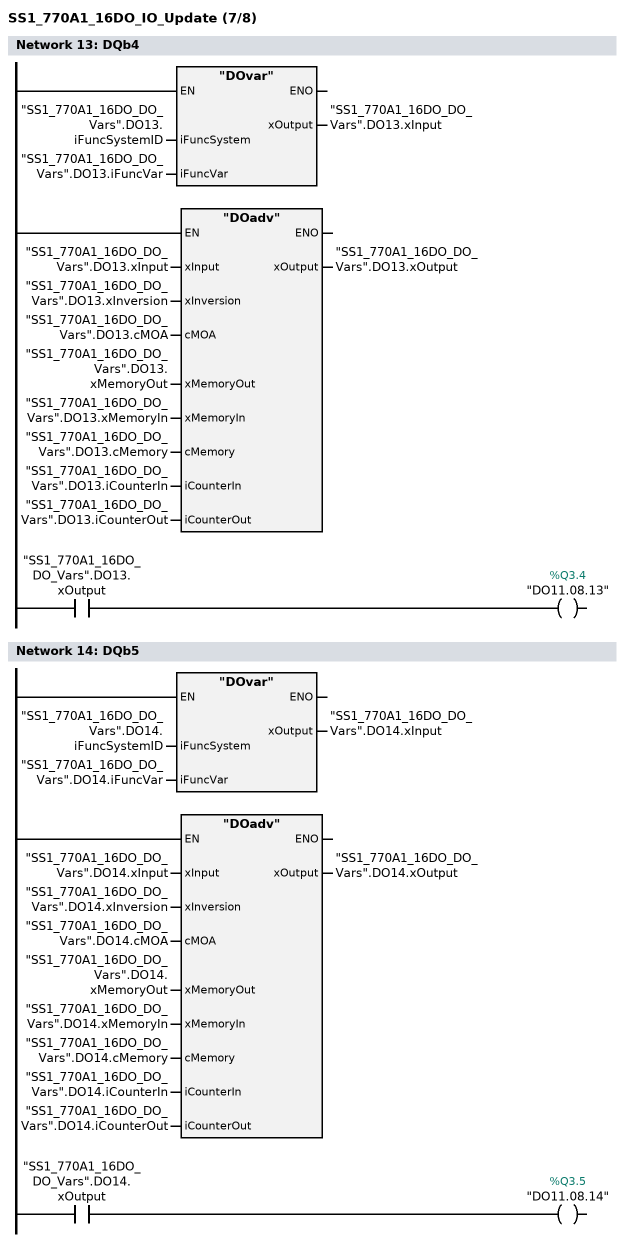
   RUNG wire#powerrail
      "DOvar"(iFuncSystem := "SS1_770A1_16DO_DO_Vars".DO13.iFuncSystemID, iFuncVar := "SS1_770A1_16DO_DO_Vars".DO13.iFuncVar, xOutput => "SS1_770A1_16DO_DO_Vars".DO13.xInput)
   END_RUNG
   RUNG wire#powerrail
      "DOadv"(xInput := "SS1_770A1_16DO_DO_Vars".DO13.xInput, xInversion := "SS1_770A1_16DO_DO_Vars".DO13.xInversion, cMOA := "SS1_770A1_16DO_DO_Vars".DO13.cMOA, xMemoryOut := "SS1_770A1_16DO_DO_Vars".DO13.xMemoryOut, xMemoryIn := "SS1_770A1_16DO_DO_Vars".DO13.xMemoryIn, cMemory := "SS1_770A1_16DO_DO_Vars".DO13.cMemory, iCounterIn := "SS1_770A1_16DO_DO_Vars".DO13.iCounterIn, iCounterOut := "SS1_770A1_16DO_DO_Vars".DO13.iCounterOut, xOutput => "SS1_770A1_16DO_DO_Vars".DO13.xOutput)
   END_RUNG
   RUNG wire#powerrail
      Contact( "SS1_770A1_16DO_DO_Vars".DO13.xOutput )
      Coil( "DO11.08.13" )
   END_RUNG
   // the same network as SCL:
   "DOvar"(iFuncSystem := "SS1_770A1_16DO_DO_Vars".DO13.iFuncSystemID,
           iFuncVar := "SS1_770A1_16DO_DO_Vars".DO13.iFuncVar,
           xOutput => "SS1_770A1_16DO_DO_Vars".DO13.xInput);
   "DOadv"(xInput := "SS1_770A1_16DO_DO_Vars".DO13.xInput,
           xInversion := "SS1_770A1_16DO_DO_Vars".DO13.xInversion,
           cMOA := "SS1_770A1_16DO_DO_Vars".DO13.cMOA,
           xMemoryOut := "SS1_770A1_16DO_DO_Vars".DO13.xMemoryOut,
           xMemoryIn := "SS1_770A1_16DO_DO_Vars".DO13.xMemoryIn,
           cMemory := "SS1_770A1_16DO_DO_Vars".DO13.cMemory,
           iCounterIn := "SS1_770A1_16DO_DO_Vars".DO13.iCounterIn,
           iCounterOut := "SS1_770A1_16DO_DO_Vars".DO13.iCounterOut,
           xOutput => "SS1_770A1_16DO_DO_Vars".DO13.xOutput);
   "DO11.08.13" := "SS1_770A1_16DO_DO_Vars".DO13.xOutput;
END_REGION

REGION Network 14: DQb5
   RUNG wire#powerrail
      "DOvar"(iFuncSystem := "SS1_770A1_16DO_DO_Vars".DO14.iFuncSystemID, iFuncVar := "SS1_770A1_16DO_DO_Vars".DO14.iFuncVar, xOutput => "SS1_770A1_16DO_DO_Vars".DO14.xInput)
   END_RUNG
   RUNG wire#powerrail
      "DOadv"(xInput := "SS1_770A1_16DO_DO_Vars".DO14.xInput, xInversion := "SS1_770A1_16DO_DO_Vars".DO14.xInversion, cMOA := "SS1_770A1_16DO_DO_Vars".DO14.cMOA, xMemoryOut := "SS1_770A1_16DO_DO_Vars".DO14.xMemoryOut, xMemoryIn := "SS1_770A1_16DO_DO_Vars".DO14.xMemoryIn, cMemory := "SS1_770A1_16DO_DO_Vars".DO14.cMemory, iCounterIn := "SS1_770A1_16DO_DO_Vars".DO14.iCounterIn, iCounterOut := "SS1_770A1_16DO_DO_Vars".DO14.iCounterOut, xOutput => "SS1_770A1_16DO_DO_Vars".DO14.xOutput)
   END_RUNG
   RUNG wire#powerrail
      Contact( "SS1_770A1_16DO_DO_Vars".DO14.xOutput )
      Coil( "DO11.08.14" )
   END_RUNG
   // the same network as SCL:
   "DOvar"(iFuncSystem := "SS1_770A1_16DO_DO_Vars".DO14.iFuncSystemID,
           iFuncVar := "SS1_770A1_16DO_DO_Vars".DO14.iFuncVar,
           xOutput => "SS1_770A1_16DO_DO_Vars".DO14.xInput);
   "DOadv"(xInput := "SS1_770A1_16DO_DO_Vars".DO14.xInput,
           xInversion := "SS1_770A1_16DO_DO_Vars".DO14.xInversion,
           cMOA := "SS1_770A1_16DO_DO_Vars".DO14.cMOA,
           xMemoryOut := "SS1_770A1_16DO_DO_Vars".DO14.xMemoryOut,
           xMemoryIn := "SS1_770A1_16DO_DO_Vars".DO14.xMemoryIn,
           cMemory := "SS1_770A1_16DO_DO_Vars".DO14.cMemory,
           iCounterIn := "SS1_770A1_16DO_DO_Vars".DO14.iCounterIn,
           iCounterOut := "SS1_770A1_16DO_DO_Vars".DO14.iCounterOut,
           xOutput => "SS1_770A1_16DO_DO_Vars".DO14.xOutput);
   "DO11.08.14" := "SS1_770A1_16DO_DO_Vars".DO14.xOutput;
END_REGION

REGION Network 15: DQb6
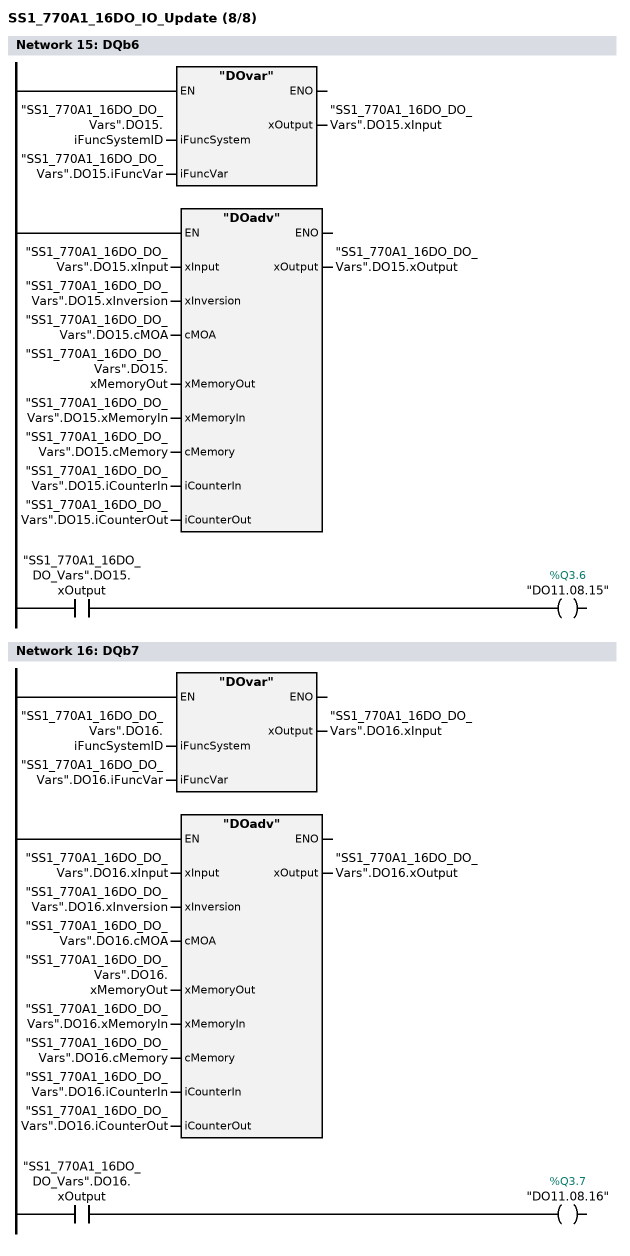
   RUNG wire#powerrail
      "DOvar"(iFuncSystem := "SS1_770A1_16DO_DO_Vars".DO15.iFuncSystemID, iFuncVar := "SS1_770A1_16DO_DO_Vars".DO15.iFuncVar, xOutput => "SS1_770A1_16DO_DO_Vars".DO15.xInput)
   END_RUNG
   RUNG wire#powerrail
      "DOadv"(xInput := "SS1_770A1_16DO_DO_Vars".DO15.xInput, xInversion := "SS1_770A1_16DO_DO_Vars".DO15.xInversion, cMOA := "SS1_770A1_16DO_DO_Vars".DO15.cMOA, xMemoryOut := "SS1_770A1_16DO_DO_Vars".DO15.xMemoryOut, xMemoryIn := "SS1_770A1_16DO_DO_Vars".DO15.xMemoryIn, cMemory := "SS1_770A1_16DO_DO_Vars".DO15.cMemory, iCounterIn := "SS1_770A1_16DO_DO_Vars".DO15.iCounterIn, iCounterOut := "SS1_770A1_16DO_DO_Vars".DO15.iCounterOut, xOutput => "SS1_770A1_16DO_DO_Vars".DO15.xOutput)
   END_RUNG
   RUNG wire#powerrail
      Contact( "SS1_770A1_16DO_DO_Vars".DO15.xOutput )
      Coil( "DO11.08.15" )
   END_RUNG
   // the same network as SCL:
   "DOvar"(iFuncSystem := "SS1_770A1_16DO_DO_Vars".DO15.iFuncSystemID,
           iFuncVar := "SS1_770A1_16DO_DO_Vars".DO15.iFuncVar,
           xOutput => "SS1_770A1_16DO_DO_Vars".DO15.xInput);
   "DOadv"(xInput := "SS1_770A1_16DO_DO_Vars".DO15.xInput,
           xInversion := "SS1_770A1_16DO_DO_Vars".DO15.xInversion,
           cMOA := "SS1_770A1_16DO_DO_Vars".DO15.cMOA,
           xMemoryOut := "SS1_770A1_16DO_DO_Vars".DO15.xMemoryOut,
           xMemoryIn := "SS1_770A1_16DO_DO_Vars".DO15.xMemoryIn,
           cMemory := "SS1_770A1_16DO_DO_Vars".DO15.cMemory,
           iCounterIn := "SS1_770A1_16DO_DO_Vars".DO15.iCounterIn,
           iCounterOut := "SS1_770A1_16DO_DO_Vars".DO15.iCounterOut,
           xOutput => "SS1_770A1_16DO_DO_Vars".DO15.xOutput);
   "DO11.08.15" := "SS1_770A1_16DO_DO_Vars".DO15.xOutput;
END_REGION

REGION Network 16: DQb7
   RUNG wire#powerrail
      "DOvar"(iFuncSystem := "SS1_770A1_16DO_DO_Vars".DO16.iFuncSystemID, iFuncVar := "SS1_770A1_16DO_DO_Vars".DO16.iFuncVar, xOutput => "SS1_770A1_16DO_DO_Vars".DO16.xInput)
   END_RUNG
   RUNG wire#powerrail
      "DOadv"(xInput := "SS1_770A1_16DO_DO_Vars".DO16.xInput, xInversion := "SS1_770A1_16DO_DO_Vars".DO16.xInversion, cMOA := "SS1_770A1_16DO_DO_Vars".DO16.cMOA, xMemoryOut := "SS1_770A1_16DO_DO_Vars".DO16.xMemoryOut, xMemoryIn := "SS1_770A1_16DO_DO_Vars".DO16.xMemoryIn, cMemory := "SS1_770A1_16DO_DO_Vars".DO16.cMemory, iCounterIn := "SS1_770A1_16DO_DO_Vars".DO16.iCounterIn, iCounterOut := "SS1_770A1_16DO_DO_Vars".DO16.iCounterOut, xOutput => "SS1_770A1_16DO_DO_Vars".DO16.xOutput)
   END_RUNG
   RUNG wire#powerrail
      Contact( "SS1_770A1_16DO_DO_Vars".DO16.xOutput )
      Coil( "DO11.08.16" )
   END_RUNG
   // the same network as SCL:
   "DOvar"(iFuncSystem := "SS1_770A1_16DO_DO_Vars".DO16.iFuncSystemID,
           iFuncVar := "SS1_770A1_16DO_DO_Vars".DO16.iFuncVar,
           xOutput => "SS1_770A1_16DO_DO_Vars".DO16.xInput);
   "DOadv"(xInput := "SS1_770A1_16DO_DO_Vars".DO16.xInput,
           xInversion := "SS1_770A1_16DO_DO_Vars".DO16.xInversion,
           cMOA := "SS1_770A1_16DO_DO_Vars".DO16.cMOA,
           xMemoryOut := "SS1_770A1_16DO_DO_Vars".DO16.xMemoryOut,
           xMemoryIn := "SS1_770A1_16DO_DO_Vars".DO16.xMemoryIn,
           cMemory := "SS1_770A1_16DO_DO_Vars".DO16.cMemory,
           iCounterIn := "SS1_770A1_16DO_DO_Vars".DO16.iCounterIn,
           iCounterOut := "SS1_770A1_16DO_DO_Vars".DO16.iCounterOut,
           xOutput => "SS1_770A1_16DO_DO_Vars".DO16.xOutput);
   "DO11.08.16" := "SS1_770A1_16DO_DO_Vars".DO16.xOutput;
END_REGION
END_FUNCTION

FUNCTION "SS1_774A1_16DO_IO_Update" : Void   // FC11070, LAD
{ S7_Optimized_Access := 'TRUE' }
VERSION : 0.1
// stored: AutoNumber false, IsIECCheckEnabled false, SetENOAutomatically false, UDAEnableTagReadback false
BEGIN

REGION Network 1: DQa0
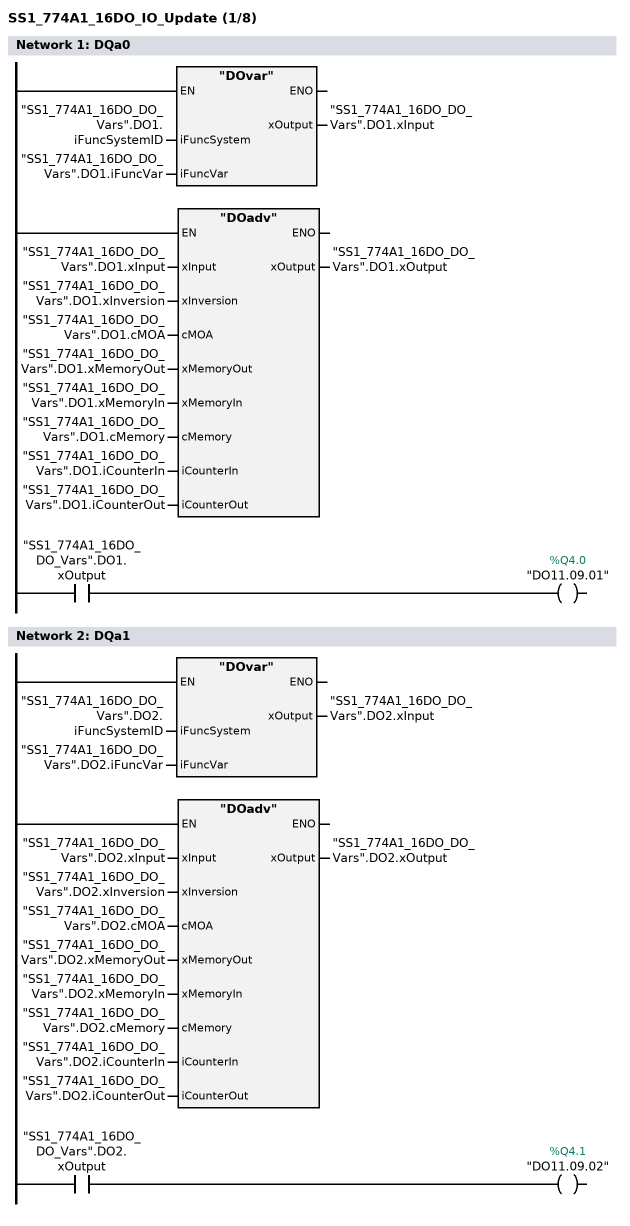
   RUNG wire#powerrail
      "DOvar"(iFuncSystem := "SS1_774A1_16DO_DO_Vars".DO1.iFuncSystemID, iFuncVar := "SS1_774A1_16DO_DO_Vars".DO1.iFuncVar, xOutput => "SS1_774A1_16DO_DO_Vars".DO1.xInput)
   END_RUNG
   RUNG wire#powerrail
      "DOadv"(xInput := "SS1_774A1_16DO_DO_Vars".DO1.xInput, xInversion := "SS1_774A1_16DO_DO_Vars".DO1.xInversion, cMOA := "SS1_774A1_16DO_DO_Vars".DO1.cMOA, xMemoryOut := "SS1_774A1_16DO_DO_Vars".DO1.xMemoryOut, xMemoryIn := "SS1_774A1_16DO_DO_Vars".DO1.xMemoryIn, cMemory := "SS1_774A1_16DO_DO_Vars".DO1.cMemory, iCounterIn := "SS1_774A1_16DO_DO_Vars".DO1.iCounterIn, iCounterOut := "SS1_774A1_16DO_DO_Vars".DO1.iCounterOut, xOutput => "SS1_774A1_16DO_DO_Vars".DO1.xOutput)
   END_RUNG
   RUNG wire#powerrail
      Contact( "SS1_774A1_16DO_DO_Vars".DO1.xOutput )
      Coil( "DO11.09.01" )
   END_RUNG
   // the same network as SCL:
   "DOvar"(iFuncSystem := "SS1_774A1_16DO_DO_Vars".DO1.iFuncSystemID,
           iFuncVar := "SS1_774A1_16DO_DO_Vars".DO1.iFuncVar,
           xOutput => "SS1_774A1_16DO_DO_Vars".DO1.xInput);
   "DOadv"(xInput := "SS1_774A1_16DO_DO_Vars".DO1.xInput,
           xInversion := "SS1_774A1_16DO_DO_Vars".DO1.xInversion,
           cMOA := "SS1_774A1_16DO_DO_Vars".DO1.cMOA,
           xMemoryOut := "SS1_774A1_16DO_DO_Vars".DO1.xMemoryOut,
           xMemoryIn := "SS1_774A1_16DO_DO_Vars".DO1.xMemoryIn,
           cMemory := "SS1_774A1_16DO_DO_Vars".DO1.cMemory,
           iCounterIn := "SS1_774A1_16DO_DO_Vars".DO1.iCounterIn,
           iCounterOut := "SS1_774A1_16DO_DO_Vars".DO1.iCounterOut,
           xOutput => "SS1_774A1_16DO_DO_Vars".DO1.xOutput);
   "DO11.09.01" := "SS1_774A1_16DO_DO_Vars".DO1.xOutput;
END_REGION

REGION Network 2: DQa1
   RUNG wire#powerrail
      "DOvar"(iFuncSystem := "SS1_774A1_16DO_DO_Vars".DO2.iFuncSystemID, iFuncVar := "SS1_774A1_16DO_DO_Vars".DO2.iFuncVar, xOutput => "SS1_774A1_16DO_DO_Vars".DO2.xInput)
   END_RUNG
   RUNG wire#powerrail
      "DOadv"(xInput := "SS1_774A1_16DO_DO_Vars".DO2.xInput, xInversion := "SS1_774A1_16DO_DO_Vars".DO2.xInversion, cMOA := "SS1_774A1_16DO_DO_Vars".DO2.cMOA, xMemoryOut := "SS1_774A1_16DO_DO_Vars".DO2.xMemoryOut, xMemoryIn := "SS1_774A1_16DO_DO_Vars".DO2.xMemoryIn, cMemory := "SS1_774A1_16DO_DO_Vars".DO2.cMemory, iCounterIn := "SS1_774A1_16DO_DO_Vars".DO2.iCounterIn, iCounterOut := "SS1_774A1_16DO_DO_Vars".DO2.iCounterOut, xOutput => "SS1_774A1_16DO_DO_Vars".DO2.xOutput)
   END_RUNG
   RUNG wire#powerrail
      Contact( "SS1_774A1_16DO_DO_Vars".DO2.xOutput )
      Coil( "DO11.09.02" )
   END_RUNG
   // the same network as SCL:
   "DOvar"(iFuncSystem := "SS1_774A1_16DO_DO_Vars".DO2.iFuncSystemID,
           iFuncVar := "SS1_774A1_16DO_DO_Vars".DO2.iFuncVar,
           xOutput => "SS1_774A1_16DO_DO_Vars".DO2.xInput);
   "DOadv"(xInput := "SS1_774A1_16DO_DO_Vars".DO2.xInput,
           xInversion := "SS1_774A1_16DO_DO_Vars".DO2.xInversion,
           cMOA := "SS1_774A1_16DO_DO_Vars".DO2.cMOA,
           xMemoryOut := "SS1_774A1_16DO_DO_Vars".DO2.xMemoryOut,
           xMemoryIn := "SS1_774A1_16DO_DO_Vars".DO2.xMemoryIn,
           cMemory := "SS1_774A1_16DO_DO_Vars".DO2.cMemory,
           iCounterIn := "SS1_774A1_16DO_DO_Vars".DO2.iCounterIn,
           iCounterOut := "SS1_774A1_16DO_DO_Vars".DO2.iCounterOut,
           xOutput => "SS1_774A1_16DO_DO_Vars".DO2.xOutput);
   "DO11.09.02" := "SS1_774A1_16DO_DO_Vars".DO2.xOutput;
END_REGION

REGION Network 3: DQa2
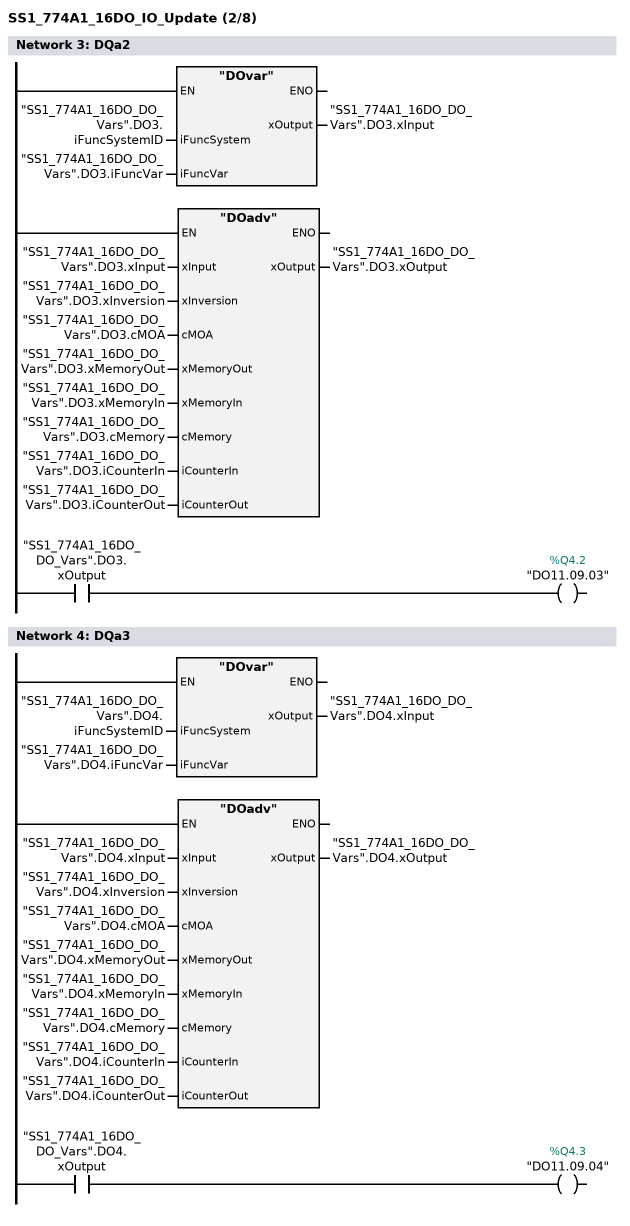
   RUNG wire#powerrail
      "DOvar"(iFuncSystem := "SS1_774A1_16DO_DO_Vars".DO3.iFuncSystemID, iFuncVar := "SS1_774A1_16DO_DO_Vars".DO3.iFuncVar, xOutput => "SS1_774A1_16DO_DO_Vars".DO3.xInput)
   END_RUNG
   RUNG wire#powerrail
      "DOadv"(xInput := "SS1_774A1_16DO_DO_Vars".DO3.xInput, xInversion := "SS1_774A1_16DO_DO_Vars".DO3.xInversion, cMOA := "SS1_774A1_16DO_DO_Vars".DO3.cMOA, xMemoryOut := "SS1_774A1_16DO_DO_Vars".DO3.xMemoryOut, xMemoryIn := "SS1_774A1_16DO_DO_Vars".DO3.xMemoryIn, cMemory := "SS1_774A1_16DO_DO_Vars".DO3.cMemory, iCounterIn := "SS1_774A1_16DO_DO_Vars".DO3.iCounterIn, iCounterOut := "SS1_774A1_16DO_DO_Vars".DO3.iCounterOut, xOutput => "SS1_774A1_16DO_DO_Vars".DO3.xOutput)
   END_RUNG
   RUNG wire#powerrail
      Contact( "SS1_774A1_16DO_DO_Vars".DO3.xOutput )
      Coil( "DO11.09.03" )
   END_RUNG
   // the same network as SCL:
   "DOvar"(iFuncSystem := "SS1_774A1_16DO_DO_Vars".DO3.iFuncSystemID,
           iFuncVar := "SS1_774A1_16DO_DO_Vars".DO3.iFuncVar,
           xOutput => "SS1_774A1_16DO_DO_Vars".DO3.xInput);
   "DOadv"(xInput := "SS1_774A1_16DO_DO_Vars".DO3.xInput,
           xInversion := "SS1_774A1_16DO_DO_Vars".DO3.xInversion,
           cMOA := "SS1_774A1_16DO_DO_Vars".DO3.cMOA,
           xMemoryOut := "SS1_774A1_16DO_DO_Vars".DO3.xMemoryOut,
           xMemoryIn := "SS1_774A1_16DO_DO_Vars".DO3.xMemoryIn,
           cMemory := "SS1_774A1_16DO_DO_Vars".DO3.cMemory,
           iCounterIn := "SS1_774A1_16DO_DO_Vars".DO3.iCounterIn,
           iCounterOut := "SS1_774A1_16DO_DO_Vars".DO3.iCounterOut,
           xOutput => "SS1_774A1_16DO_DO_Vars".DO3.xOutput);
   "DO11.09.03" := "SS1_774A1_16DO_DO_Vars".DO3.xOutput;
END_REGION

REGION Network 4: DQa3
   RUNG wire#powerrail
      "DOvar"(iFuncSystem := "SS1_774A1_16DO_DO_Vars".DO4.iFuncSystemID, iFuncVar := "SS1_774A1_16DO_DO_Vars".DO4.iFuncVar, xOutput => "SS1_774A1_16DO_DO_Vars".DO4.xInput)
   END_RUNG
   RUNG wire#powerrail
      "DOadv"(xInput := "SS1_774A1_16DO_DO_Vars".DO4.xInput, xInversion := "SS1_774A1_16DO_DO_Vars".DO4.xInversion, cMOA := "SS1_774A1_16DO_DO_Vars".DO4.cMOA, xMemoryOut := "SS1_774A1_16DO_DO_Vars".DO4.xMemoryOut, xMemoryIn := "SS1_774A1_16DO_DO_Vars".DO4.xMemoryIn, cMemory := "SS1_774A1_16DO_DO_Vars".DO4.cMemory, iCounterIn := "SS1_774A1_16DO_DO_Vars".DO4.iCounterIn, iCounterOut := "SS1_774A1_16DO_DO_Vars".DO4.iCounterOut, xOutput => "SS1_774A1_16DO_DO_Vars".DO4.xOutput)
   END_RUNG
   RUNG wire#powerrail
      Contact( "SS1_774A1_16DO_DO_Vars".DO4.xOutput )
      Coil( "DO11.09.04" )
   END_RUNG
   // the same network as SCL:
   "DOvar"(iFuncSystem := "SS1_774A1_16DO_DO_Vars".DO4.iFuncSystemID,
           iFuncVar := "SS1_774A1_16DO_DO_Vars".DO4.iFuncVar,
           xOutput => "SS1_774A1_16DO_DO_Vars".DO4.xInput);
   "DOadv"(xInput := "SS1_774A1_16DO_DO_Vars".DO4.xInput,
           xInversion := "SS1_774A1_16DO_DO_Vars".DO4.xInversion,
           cMOA := "SS1_774A1_16DO_DO_Vars".DO4.cMOA,
           xMemoryOut := "SS1_774A1_16DO_DO_Vars".DO4.xMemoryOut,
           xMemoryIn := "SS1_774A1_16DO_DO_Vars".DO4.xMemoryIn,
           cMemory := "SS1_774A1_16DO_DO_Vars".DO4.cMemory,
           iCounterIn := "SS1_774A1_16DO_DO_Vars".DO4.iCounterIn,
           iCounterOut := "SS1_774A1_16DO_DO_Vars".DO4.iCounterOut,
           xOutput => "SS1_774A1_16DO_DO_Vars".DO4.xOutput);
   "DO11.09.04" := "SS1_774A1_16DO_DO_Vars".DO4.xOutput;
END_REGION

REGION Network 5: DQa4
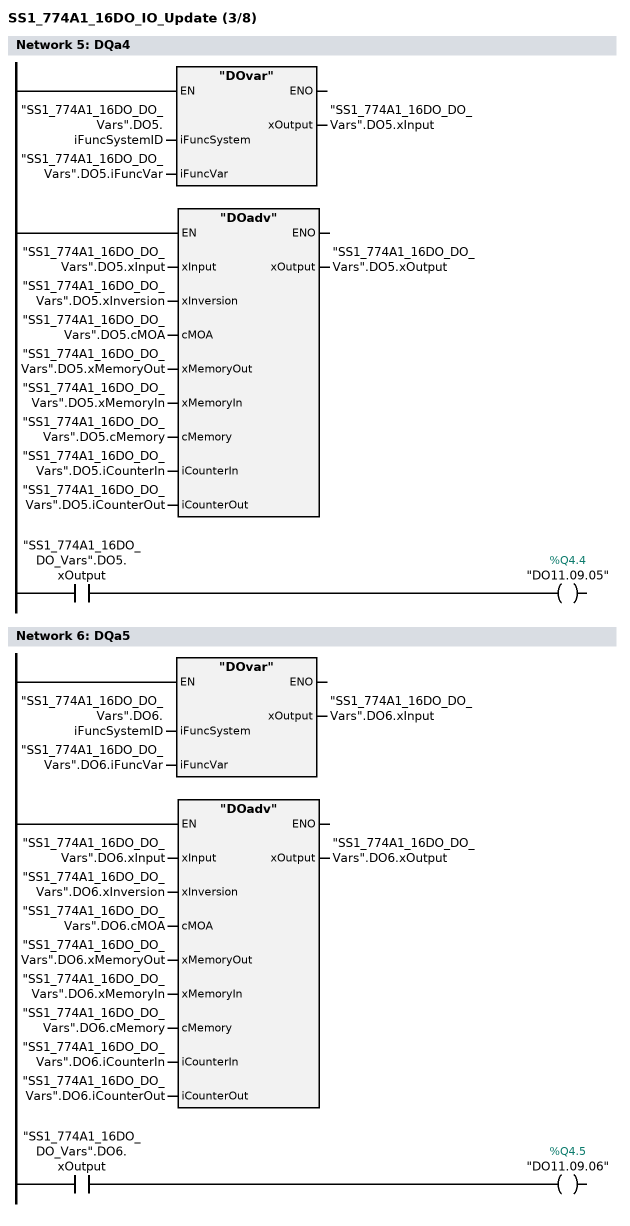
   RUNG wire#powerrail
      "DOvar"(iFuncSystem := "SS1_774A1_16DO_DO_Vars".DO5.iFuncSystemID, iFuncVar := "SS1_774A1_16DO_DO_Vars".DO5.iFuncVar, xOutput => "SS1_774A1_16DO_DO_Vars".DO5.xInput)
   END_RUNG
   RUNG wire#powerrail
      "DOadv"(xInput := "SS1_774A1_16DO_DO_Vars".DO5.xInput, xInversion := "SS1_774A1_16DO_DO_Vars".DO5.xInversion, cMOA := "SS1_774A1_16DO_DO_Vars".DO5.cMOA, xMemoryOut := "SS1_774A1_16DO_DO_Vars".DO5.xMemoryOut, xMemoryIn := "SS1_774A1_16DO_DO_Vars".DO5.xMemoryIn, cMemory := "SS1_774A1_16DO_DO_Vars".DO5.cMemory, iCounterIn := "SS1_774A1_16DO_DO_Vars".DO5.iCounterIn, iCounterOut := "SS1_774A1_16DO_DO_Vars".DO5.iCounterOut, xOutput => "SS1_774A1_16DO_DO_Vars".DO5.xOutput)
   END_RUNG
   RUNG wire#powerrail
      Contact( "SS1_774A1_16DO_DO_Vars".DO5.xOutput )
      Coil( "DO11.09.05" )
   END_RUNG
   // the same network as SCL:
   "DOvar"(iFuncSystem := "SS1_774A1_16DO_DO_Vars".DO5.iFuncSystemID,
           iFuncVar := "SS1_774A1_16DO_DO_Vars".DO5.iFuncVar,
           xOutput => "SS1_774A1_16DO_DO_Vars".DO5.xInput);
   "DOadv"(xInput := "SS1_774A1_16DO_DO_Vars".DO5.xInput,
           xInversion := "SS1_774A1_16DO_DO_Vars".DO5.xInversion,
           cMOA := "SS1_774A1_16DO_DO_Vars".DO5.cMOA,
           xMemoryOut := "SS1_774A1_16DO_DO_Vars".DO5.xMemoryOut,
           xMemoryIn := "SS1_774A1_16DO_DO_Vars".DO5.xMemoryIn,
           cMemory := "SS1_774A1_16DO_DO_Vars".DO5.cMemory,
           iCounterIn := "SS1_774A1_16DO_DO_Vars".DO5.iCounterIn,
           iCounterOut := "SS1_774A1_16DO_DO_Vars".DO5.iCounterOut,
           xOutput => "SS1_774A1_16DO_DO_Vars".DO5.xOutput);
   "DO11.09.05" := "SS1_774A1_16DO_DO_Vars".DO5.xOutput;
END_REGION

REGION Network 6: DQa5
   RUNG wire#powerrail
      "DOvar"(iFuncSystem := "SS1_774A1_16DO_DO_Vars".DO6.iFuncSystemID, iFuncVar := "SS1_774A1_16DO_DO_Vars".DO6.iFuncVar, xOutput => "SS1_774A1_16DO_DO_Vars".DO6.xInput)
   END_RUNG
   RUNG wire#powerrail
      "DOadv"(xInput := "SS1_774A1_16DO_DO_Vars".DO6.xInput, xInversion := "SS1_774A1_16DO_DO_Vars".DO6.xInversion, cMOA := "SS1_774A1_16DO_DO_Vars".DO6.cMOA, xMemoryOut := "SS1_774A1_16DO_DO_Vars".DO6.xMemoryOut, xMemoryIn := "SS1_774A1_16DO_DO_Vars".DO6.xMemoryIn, cMemory := "SS1_774A1_16DO_DO_Vars".DO6.cMemory, iCounterIn := "SS1_774A1_16DO_DO_Vars".DO6.iCounterIn, iCounterOut := "SS1_774A1_16DO_DO_Vars".DO6.iCounterOut, xOutput => "SS1_774A1_16DO_DO_Vars".DO6.xOutput)
   END_RUNG
   RUNG wire#powerrail
      Contact( "SS1_774A1_16DO_DO_Vars".DO6.xOutput )
      Coil( "DO11.09.06" )
   END_RUNG
   // the same network as SCL:
   "DOvar"(iFuncSystem := "SS1_774A1_16DO_DO_Vars".DO6.iFuncSystemID,
           iFuncVar := "SS1_774A1_16DO_DO_Vars".DO6.iFuncVar,
           xOutput => "SS1_774A1_16DO_DO_Vars".DO6.xInput);
   "DOadv"(xInput := "SS1_774A1_16DO_DO_Vars".DO6.xInput,
           xInversion := "SS1_774A1_16DO_DO_Vars".DO6.xInversion,
           cMOA := "SS1_774A1_16DO_DO_Vars".DO6.cMOA,
           xMemoryOut := "SS1_774A1_16DO_DO_Vars".DO6.xMemoryOut,
           xMemoryIn := "SS1_774A1_16DO_DO_Vars".DO6.xMemoryIn,
           cMemory := "SS1_774A1_16DO_DO_Vars".DO6.cMemory,
           iCounterIn := "SS1_774A1_16DO_DO_Vars".DO6.iCounterIn,
           iCounterOut := "SS1_774A1_16DO_DO_Vars".DO6.iCounterOut,
           xOutput => "SS1_774A1_16DO_DO_Vars".DO6.xOutput);
   "DO11.09.06" := "SS1_774A1_16DO_DO_Vars".DO6.xOutput;
END_REGION

REGION Network 7: DQa6
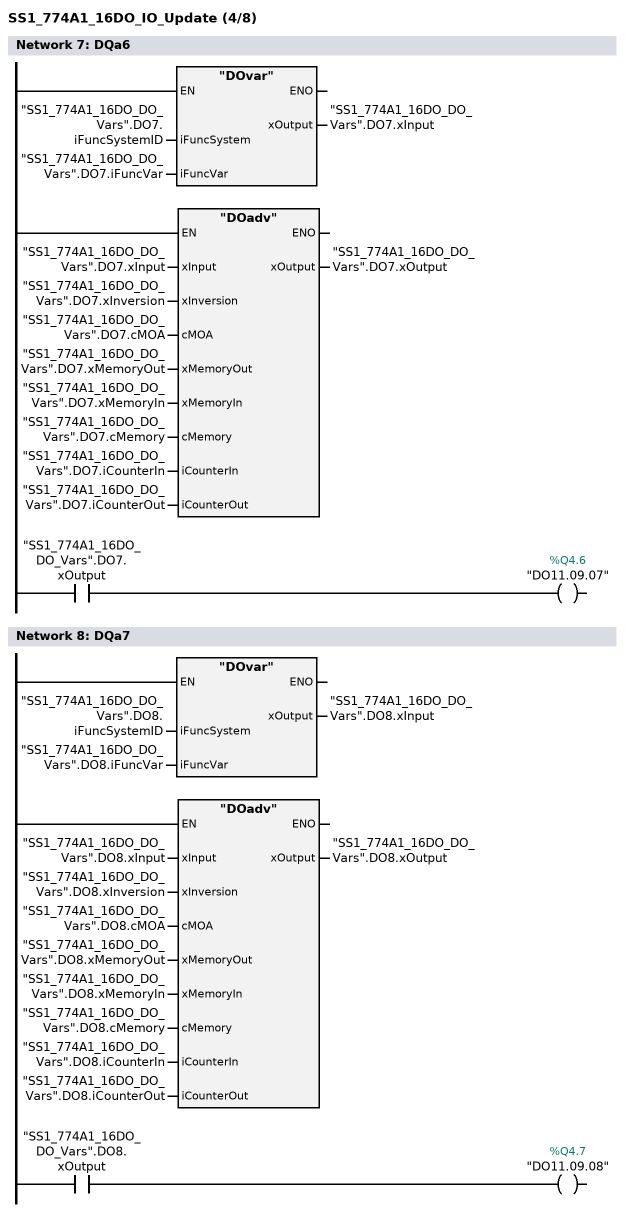
   RUNG wire#powerrail
      "DOvar"(iFuncSystem := "SS1_774A1_16DO_DO_Vars".DO7.iFuncSystemID, iFuncVar := "SS1_774A1_16DO_DO_Vars".DO7.iFuncVar, xOutput => "SS1_774A1_16DO_DO_Vars".DO7.xInput)
   END_RUNG
   RUNG wire#powerrail
      "DOadv"(xInput := "SS1_774A1_16DO_DO_Vars".DO7.xInput, xInversion := "SS1_774A1_16DO_DO_Vars".DO7.xInversion, cMOA := "SS1_774A1_16DO_DO_Vars".DO7.cMOA, xMemoryOut := "SS1_774A1_16DO_DO_Vars".DO7.xMemoryOut, xMemoryIn := "SS1_774A1_16DO_DO_Vars".DO7.xMemoryIn, cMemory := "SS1_774A1_16DO_DO_Vars".DO7.cMemory, iCounterIn := "SS1_774A1_16DO_DO_Vars".DO7.iCounterIn, iCounterOut := "SS1_774A1_16DO_DO_Vars".DO7.iCounterOut, xOutput => "SS1_774A1_16DO_DO_Vars".DO7.xOutput)
   END_RUNG
   RUNG wire#powerrail
      Contact( "SS1_774A1_16DO_DO_Vars".DO7.xOutput )
      Coil( "DO11.09.07" )
   END_RUNG
   // the same network as SCL:
   "DOvar"(iFuncSystem := "SS1_774A1_16DO_DO_Vars".DO7.iFuncSystemID,
           iFuncVar := "SS1_774A1_16DO_DO_Vars".DO7.iFuncVar,
           xOutput => "SS1_774A1_16DO_DO_Vars".DO7.xInput);
   "DOadv"(xInput := "SS1_774A1_16DO_DO_Vars".DO7.xInput,
           xInversion := "SS1_774A1_16DO_DO_Vars".DO7.xInversion,
           cMOA := "SS1_774A1_16DO_DO_Vars".DO7.cMOA,
           xMemoryOut := "SS1_774A1_16DO_DO_Vars".DO7.xMemoryOut,
           xMemoryIn := "SS1_774A1_16DO_DO_Vars".DO7.xMemoryIn,
           cMemory := "SS1_774A1_16DO_DO_Vars".DO7.cMemory,
           iCounterIn := "SS1_774A1_16DO_DO_Vars".DO7.iCounterIn,
           iCounterOut := "SS1_774A1_16DO_DO_Vars".DO7.iCounterOut,
           xOutput => "SS1_774A1_16DO_DO_Vars".DO7.xOutput);
   "DO11.09.07" := "SS1_774A1_16DO_DO_Vars".DO7.xOutput;
END_REGION

REGION Network 8: DQa7
   RUNG wire#powerrail
      "DOvar"(iFuncSystem := "SS1_774A1_16DO_DO_Vars".DO8.iFuncSystemID, iFuncVar := "SS1_774A1_16DO_DO_Vars".DO8.iFuncVar, xOutput => "SS1_774A1_16DO_DO_Vars".DO8.xInput)
   END_RUNG
   RUNG wire#powerrail
      "DOadv"(xInput := "SS1_774A1_16DO_DO_Vars".DO8.xInput, xInversion := "SS1_774A1_16DO_DO_Vars".DO8.xInversion, cMOA := "SS1_774A1_16DO_DO_Vars".DO8.cMOA, xMemoryOut := "SS1_774A1_16DO_DO_Vars".DO8.xMemoryOut, xMemoryIn := "SS1_774A1_16DO_DO_Vars".DO8.xMemoryIn, cMemory := "SS1_774A1_16DO_DO_Vars".DO8.cMemory, iCounterIn := "SS1_774A1_16DO_DO_Vars".DO8.iCounterIn, iCounterOut := "SS1_774A1_16DO_DO_Vars".DO8.iCounterOut, xOutput => "SS1_774A1_16DO_DO_Vars".DO8.xOutput)
   END_RUNG
   RUNG wire#powerrail
      Contact( "SS1_774A1_16DO_DO_Vars".DO8.xOutput )
      Coil( "DO11.09.08" )
   END_RUNG
   // the same network as SCL:
   "DOvar"(iFuncSystem := "SS1_774A1_16DO_DO_Vars".DO8.iFuncSystemID,
           iFuncVar := "SS1_774A1_16DO_DO_Vars".DO8.iFuncVar,
           xOutput => "SS1_774A1_16DO_DO_Vars".DO8.xInput);
   "DOadv"(xInput := "SS1_774A1_16DO_DO_Vars".DO8.xInput,
           xInversion := "SS1_774A1_16DO_DO_Vars".DO8.xInversion,
           cMOA := "SS1_774A1_16DO_DO_Vars".DO8.cMOA,
           xMemoryOut := "SS1_774A1_16DO_DO_Vars".DO8.xMemoryOut,
           xMemoryIn := "SS1_774A1_16DO_DO_Vars".DO8.xMemoryIn,
           cMemory := "SS1_774A1_16DO_DO_Vars".DO8.cMemory,
           iCounterIn := "SS1_774A1_16DO_DO_Vars".DO8.iCounterIn,
           iCounterOut := "SS1_774A1_16DO_DO_Vars".DO8.iCounterOut,
           xOutput => "SS1_774A1_16DO_DO_Vars".DO8.xOutput);
   "DO11.09.08" := "SS1_774A1_16DO_DO_Vars".DO8.xOutput;
END_REGION

REGION Network 9: DQb0
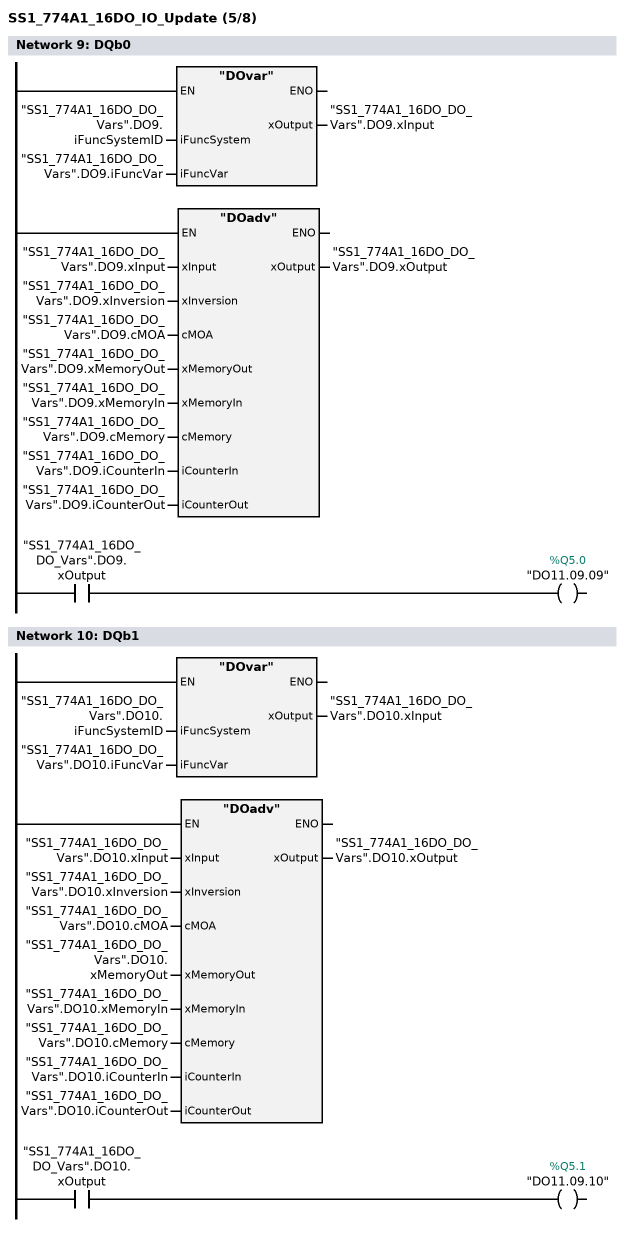
   RUNG wire#powerrail
      "DOvar"(iFuncSystem := "SS1_774A1_16DO_DO_Vars".DO9.iFuncSystemID, iFuncVar := "SS1_774A1_16DO_DO_Vars".DO9.iFuncVar, xOutput => "SS1_774A1_16DO_DO_Vars".DO9.xInput)
   END_RUNG
   RUNG wire#powerrail
      "DOadv"(xInput := "SS1_774A1_16DO_DO_Vars".DO9.xInput, xInversion := "SS1_774A1_16DO_DO_Vars".DO9.xInversion, cMOA := "SS1_774A1_16DO_DO_Vars".DO9.cMOA, xMemoryOut := "SS1_774A1_16DO_DO_Vars".DO9.xMemoryOut, xMemoryIn := "SS1_774A1_16DO_DO_Vars".DO9.xMemoryIn, cMemory := "SS1_774A1_16DO_DO_Vars".DO9.cMemory, iCounterIn := "SS1_774A1_16DO_DO_Vars".DO9.iCounterIn, iCounterOut := "SS1_774A1_16DO_DO_Vars".DO9.iCounterOut, xOutput => "SS1_774A1_16DO_DO_Vars".DO9.xOutput)
   END_RUNG
   RUNG wire#powerrail
      Contact( "SS1_774A1_16DO_DO_Vars".DO9.xOutput )
      Coil( "DO11.09.09" )
   END_RUNG
   // the same network as SCL:
   "DOvar"(iFuncSystem := "SS1_774A1_16DO_DO_Vars".DO9.iFuncSystemID,
           iFuncVar := "SS1_774A1_16DO_DO_Vars".DO9.iFuncVar,
           xOutput => "SS1_774A1_16DO_DO_Vars".DO9.xInput);
   "DOadv"(xInput := "SS1_774A1_16DO_DO_Vars".DO9.xInput,
           xInversion := "SS1_774A1_16DO_DO_Vars".DO9.xInversion,
           cMOA := "SS1_774A1_16DO_DO_Vars".DO9.cMOA,
           xMemoryOut := "SS1_774A1_16DO_DO_Vars".DO9.xMemoryOut,
           xMemoryIn := "SS1_774A1_16DO_DO_Vars".DO9.xMemoryIn,
           cMemory := "SS1_774A1_16DO_DO_Vars".DO9.cMemory,
           iCounterIn := "SS1_774A1_16DO_DO_Vars".DO9.iCounterIn,
           iCounterOut := "SS1_774A1_16DO_DO_Vars".DO9.iCounterOut,
           xOutput => "SS1_774A1_16DO_DO_Vars".DO9.xOutput);
   "DO11.09.09" := "SS1_774A1_16DO_DO_Vars".DO9.xOutput;
END_REGION

REGION Network 10: DQb1
   RUNG wire#powerrail
      "DOvar"(iFuncSystem := "SS1_774A1_16DO_DO_Vars".DO10.iFuncSystemID, iFuncVar := "SS1_774A1_16DO_DO_Vars".DO10.iFuncVar, xOutput => "SS1_774A1_16DO_DO_Vars".DO10.xInput)
   END_RUNG
   RUNG wire#powerrail
      "DOadv"(xInput := "SS1_774A1_16DO_DO_Vars".DO10.xInput, xInversion := "SS1_774A1_16DO_DO_Vars".DO10.xInversion, cMOA := "SS1_774A1_16DO_DO_Vars".DO10.cMOA, xMemoryOut := "SS1_774A1_16DO_DO_Vars".DO10.xMemoryOut, xMemoryIn := "SS1_774A1_16DO_DO_Vars".DO10.xMemoryIn, cMemory := "SS1_774A1_16DO_DO_Vars".DO10.cMemory, iCounterIn := "SS1_774A1_16DO_DO_Vars".DO10.iCounterIn, iCounterOut := "SS1_774A1_16DO_DO_Vars".DO10.iCounterOut, xOutput => "SS1_774A1_16DO_DO_Vars".DO10.xOutput)
   END_RUNG
   RUNG wire#powerrail
      Contact( "SS1_774A1_16DO_DO_Vars".DO10.xOutput )
      Coil( "DO11.09.10" )
   END_RUNG
   // the same network as SCL:
   "DOvar"(iFuncSystem := "SS1_774A1_16DO_DO_Vars".DO10.iFuncSystemID,
           iFuncVar := "SS1_774A1_16DO_DO_Vars".DO10.iFuncVar,
           xOutput => "SS1_774A1_16DO_DO_Vars".DO10.xInput);
   "DOadv"(xInput := "SS1_774A1_16DO_DO_Vars".DO10.xInput,
           xInversion := "SS1_774A1_16DO_DO_Vars".DO10.xInversion,
           cMOA := "SS1_774A1_16DO_DO_Vars".DO10.cMOA,
           xMemoryOut := "SS1_774A1_16DO_DO_Vars".DO10.xMemoryOut,
           xMemoryIn := "SS1_774A1_16DO_DO_Vars".DO10.xMemoryIn,
           cMemory := "SS1_774A1_16DO_DO_Vars".DO10.cMemory,
           iCounterIn := "SS1_774A1_16DO_DO_Vars".DO10.iCounterIn,
           iCounterOut := "SS1_774A1_16DO_DO_Vars".DO10.iCounterOut,
           xOutput => "SS1_774A1_16DO_DO_Vars".DO10.xOutput);
   "DO11.09.10" := "SS1_774A1_16DO_DO_Vars".DO10.xOutput;
END_REGION

REGION Network 11: DQb2
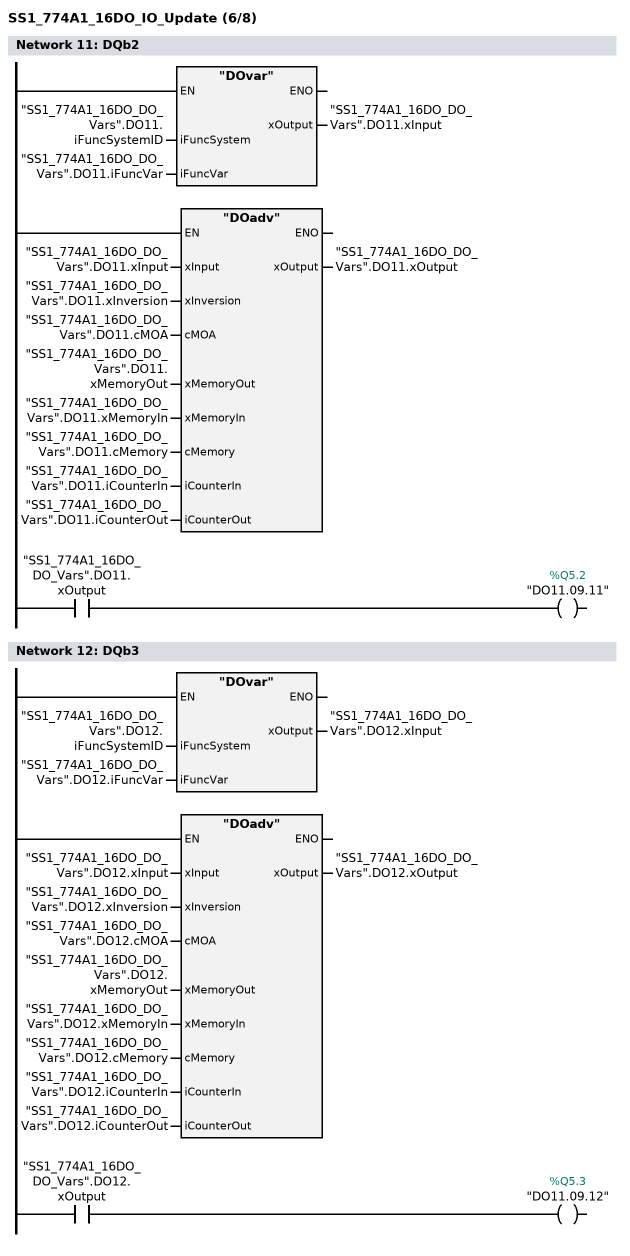
   RUNG wire#powerrail
      "DOvar"(iFuncSystem := "SS1_774A1_16DO_DO_Vars".DO11.iFuncSystemID, iFuncVar := "SS1_774A1_16DO_DO_Vars".DO11.iFuncVar, xOutput => "SS1_774A1_16DO_DO_Vars".DO11.xInput)
   END_RUNG
   RUNG wire#powerrail
      "DOadv"(xInput := "SS1_774A1_16DO_DO_Vars".DO11.xInput, xInversion := "SS1_774A1_16DO_DO_Vars".DO11.xInversion, cMOA := "SS1_774A1_16DO_DO_Vars".DO11.cMOA, xMemoryOut := "SS1_774A1_16DO_DO_Vars".DO11.xMemoryOut, xMemoryIn := "SS1_774A1_16DO_DO_Vars".DO11.xMemoryIn, cMemory := "SS1_774A1_16DO_DO_Vars".DO11.cMemory, iCounterIn := "SS1_774A1_16DO_DO_Vars".DO11.iCounterIn, iCounterOut := "SS1_774A1_16DO_DO_Vars".DO11.iCounterOut, xOutput => "SS1_774A1_16DO_DO_Vars".DO11.xOutput)
   END_RUNG
   RUNG wire#powerrail
      Contact( "SS1_774A1_16DO_DO_Vars".DO11.xOutput )
      Coil( "DO11.09.11" )
   END_RUNG
   // the same network as SCL:
   "DOvar"(iFuncSystem := "SS1_774A1_16DO_DO_Vars".DO11.iFuncSystemID,
           iFuncVar := "SS1_774A1_16DO_DO_Vars".DO11.iFuncVar,
           xOutput => "SS1_774A1_16DO_DO_Vars".DO11.xInput);
   "DOadv"(xInput := "SS1_774A1_16DO_DO_Vars".DO11.xInput,
           xInversion := "SS1_774A1_16DO_DO_Vars".DO11.xInversion,
           cMOA := "SS1_774A1_16DO_DO_Vars".DO11.cMOA,
           xMemoryOut := "SS1_774A1_16DO_DO_Vars".DO11.xMemoryOut,
           xMemoryIn := "SS1_774A1_16DO_DO_Vars".DO11.xMemoryIn,
           cMemory := "SS1_774A1_16DO_DO_Vars".DO11.cMemory,
           iCounterIn := "SS1_774A1_16DO_DO_Vars".DO11.iCounterIn,
           iCounterOut := "SS1_774A1_16DO_DO_Vars".DO11.iCounterOut,
           xOutput => "SS1_774A1_16DO_DO_Vars".DO11.xOutput);
   "DO11.09.11" := "SS1_774A1_16DO_DO_Vars".DO11.xOutput;
END_REGION

REGION Network 12: DQb3
   RUNG wire#powerrail
      "DOvar"(iFuncSystem := "SS1_774A1_16DO_DO_Vars".DO12.iFuncSystemID, iFuncVar := "SS1_774A1_16DO_DO_Vars".DO12.iFuncVar, xOutput => "SS1_774A1_16DO_DO_Vars".DO12.xInput)
   END_RUNG
   RUNG wire#powerrail
      "DOadv"(xInput := "SS1_774A1_16DO_DO_Vars".DO12.xInput, xInversion := "SS1_774A1_16DO_DO_Vars".DO12.xInversion, cMOA := "SS1_774A1_16DO_DO_Vars".DO12.cMOA, xMemoryOut := "SS1_774A1_16DO_DO_Vars".DO12.xMemoryOut, xMemoryIn := "SS1_774A1_16DO_DO_Vars".DO12.xMemoryIn, cMemory := "SS1_774A1_16DO_DO_Vars".DO12.cMemory, iCounterIn := "SS1_774A1_16DO_DO_Vars".DO12.iCounterIn, iCounterOut := "SS1_774A1_16DO_DO_Vars".DO12.iCounterOut, xOutput => "SS1_774A1_16DO_DO_Vars".DO12.xOutput)
   END_RUNG
   RUNG wire#powerrail
      Contact( "SS1_774A1_16DO_DO_Vars".DO12.xOutput )
      Coil( "DO11.09.12" )
   END_RUNG
   // the same network as SCL:
   "DOvar"(iFuncSystem := "SS1_774A1_16DO_DO_Vars".DO12.iFuncSystemID,
           iFuncVar := "SS1_774A1_16DO_DO_Vars".DO12.iFuncVar,
           xOutput => "SS1_774A1_16DO_DO_Vars".DO12.xInput);
   "DOadv"(xInput := "SS1_774A1_16DO_DO_Vars".DO12.xInput,
           xInversion := "SS1_774A1_16DO_DO_Vars".DO12.xInversion,
           cMOA := "SS1_774A1_16DO_DO_Vars".DO12.cMOA,
           xMemoryOut := "SS1_774A1_16DO_DO_Vars".DO12.xMemoryOut,
           xMemoryIn := "SS1_774A1_16DO_DO_Vars".DO12.xMemoryIn,
           cMemory := "SS1_774A1_16DO_DO_Vars".DO12.cMemory,
           iCounterIn := "SS1_774A1_16DO_DO_Vars".DO12.iCounterIn,
           iCounterOut := "SS1_774A1_16DO_DO_Vars".DO12.iCounterOut,
           xOutput => "SS1_774A1_16DO_DO_Vars".DO12.xOutput);
   "DO11.09.12" := "SS1_774A1_16DO_DO_Vars".DO12.xOutput;
END_REGION

REGION Network 13: DQb4
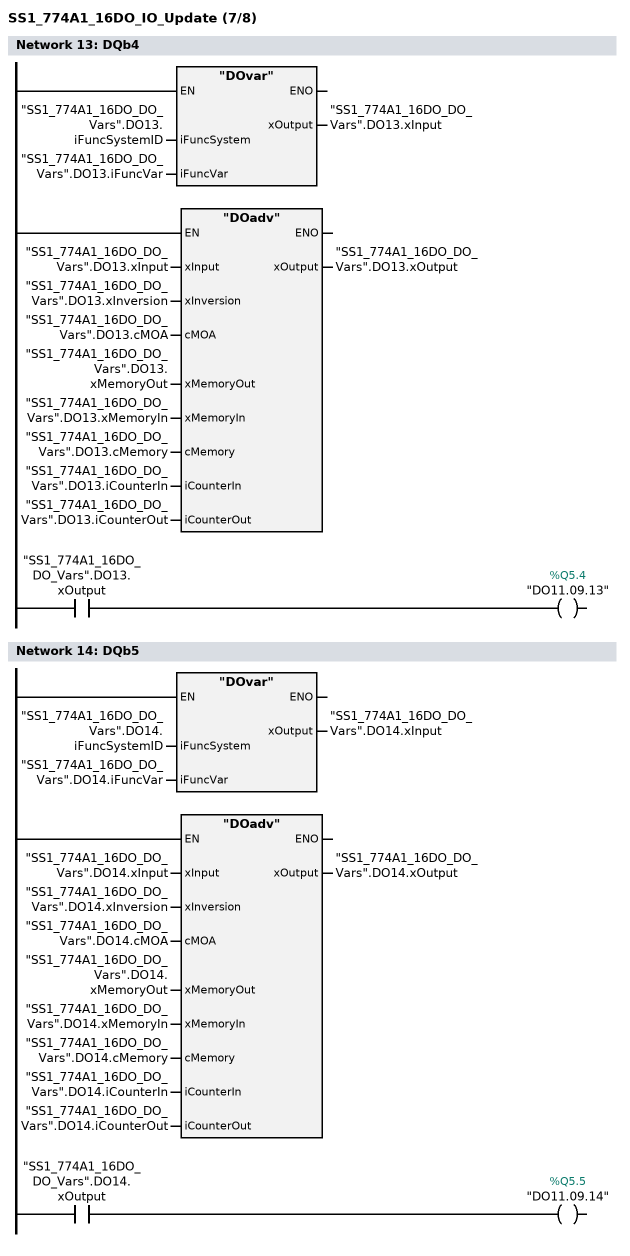
   RUNG wire#powerrail
      "DOvar"(iFuncSystem := "SS1_774A1_16DO_DO_Vars".DO13.iFuncSystemID, iFuncVar := "SS1_774A1_16DO_DO_Vars".DO13.iFuncVar, xOutput => "SS1_774A1_16DO_DO_Vars".DO13.xInput)
   END_RUNG
   RUNG wire#powerrail
      "DOadv"(xInput := "SS1_774A1_16DO_DO_Vars".DO13.xInput, xInversion := "SS1_774A1_16DO_DO_Vars".DO13.xInversion, cMOA := "SS1_774A1_16DO_DO_Vars".DO13.cMOA, xMemoryOut := "SS1_774A1_16DO_DO_Vars".DO13.xMemoryOut, xMemoryIn := "SS1_774A1_16DO_DO_Vars".DO13.xMemoryIn, cMemory := "SS1_774A1_16DO_DO_Vars".DO13.cMemory, iCounterIn := "SS1_774A1_16DO_DO_Vars".DO13.iCounterIn, iCounterOut := "SS1_774A1_16DO_DO_Vars".DO13.iCounterOut, xOutput => "SS1_774A1_16DO_DO_Vars".DO13.xOutput)
   END_RUNG
   RUNG wire#powerrail
      Contact( "SS1_774A1_16DO_DO_Vars".DO13.xOutput )
      Coil( "DO11.09.13" )
   END_RUNG
   // the same network as SCL:
   "DOvar"(iFuncSystem := "SS1_774A1_16DO_DO_Vars".DO13.iFuncSystemID,
           iFuncVar := "SS1_774A1_16DO_DO_Vars".DO13.iFuncVar,
           xOutput => "SS1_774A1_16DO_DO_Vars".DO13.xInput);
   "DOadv"(xInput := "SS1_774A1_16DO_DO_Vars".DO13.xInput,
           xInversion := "SS1_774A1_16DO_DO_Vars".DO13.xInversion,
           cMOA := "SS1_774A1_16DO_DO_Vars".DO13.cMOA,
           xMemoryOut := "SS1_774A1_16DO_DO_Vars".DO13.xMemoryOut,
           xMemoryIn := "SS1_774A1_16DO_DO_Vars".DO13.xMemoryIn,
           cMemory := "SS1_774A1_16DO_DO_Vars".DO13.cMemory,
           iCounterIn := "SS1_774A1_16DO_DO_Vars".DO13.iCounterIn,
           iCounterOut := "SS1_774A1_16DO_DO_Vars".DO13.iCounterOut,
           xOutput => "SS1_774A1_16DO_DO_Vars".DO13.xOutput);
   "DO11.09.13" := "SS1_774A1_16DO_DO_Vars".DO13.xOutput;
END_REGION

REGION Network 14: DQb5
   RUNG wire#powerrail
      "DOvar"(iFuncSystem := "SS1_774A1_16DO_DO_Vars".DO14.iFuncSystemID, iFuncVar := "SS1_774A1_16DO_DO_Vars".DO14.iFuncVar, xOutput => "SS1_774A1_16DO_DO_Vars".DO14.xInput)
   END_RUNG
   RUNG wire#powerrail
      "DOadv"(xInput := "SS1_774A1_16DO_DO_Vars".DO14.xInput, xInversion := "SS1_774A1_16DO_DO_Vars".DO14.xInversion, cMOA := "SS1_774A1_16DO_DO_Vars".DO14.cMOA, xMemoryOut := "SS1_774A1_16DO_DO_Vars".DO14.xMemoryOut, xMemoryIn := "SS1_774A1_16DO_DO_Vars".DO14.xMemoryIn, cMemory := "SS1_774A1_16DO_DO_Vars".DO14.cMemory, iCounterIn := "SS1_774A1_16DO_DO_Vars".DO14.iCounterIn, iCounterOut := "SS1_774A1_16DO_DO_Vars".DO14.iCounterOut, xOutput => "SS1_774A1_16DO_DO_Vars".DO14.xOutput)
   END_RUNG
   RUNG wire#powerrail
      Contact( "SS1_774A1_16DO_DO_Vars".DO14.xOutput )
      Coil( "DO11.09.14" )
   END_RUNG
   // the same network as SCL:
   "DOvar"(iFuncSystem := "SS1_774A1_16DO_DO_Vars".DO14.iFuncSystemID,
           iFuncVar := "SS1_774A1_16DO_DO_Vars".DO14.iFuncVar,
           xOutput => "SS1_774A1_16DO_DO_Vars".DO14.xInput);
   "DOadv"(xInput := "SS1_774A1_16DO_DO_Vars".DO14.xInput,
           xInversion := "SS1_774A1_16DO_DO_Vars".DO14.xInversion,
           cMOA := "SS1_774A1_16DO_DO_Vars".DO14.cMOA,
           xMemoryOut := "SS1_774A1_16DO_DO_Vars".DO14.xMemoryOut,
           xMemoryIn := "SS1_774A1_16DO_DO_Vars".DO14.xMemoryIn,
           cMemory := "SS1_774A1_16DO_DO_Vars".DO14.cMemory,
           iCounterIn := "SS1_774A1_16DO_DO_Vars".DO14.iCounterIn,
           iCounterOut := "SS1_774A1_16DO_DO_Vars".DO14.iCounterOut,
           xOutput => "SS1_774A1_16DO_DO_Vars".DO14.xOutput);
   "DO11.09.14" := "SS1_774A1_16DO_DO_Vars".DO14.xOutput;
END_REGION

REGION Network 15: DQb6
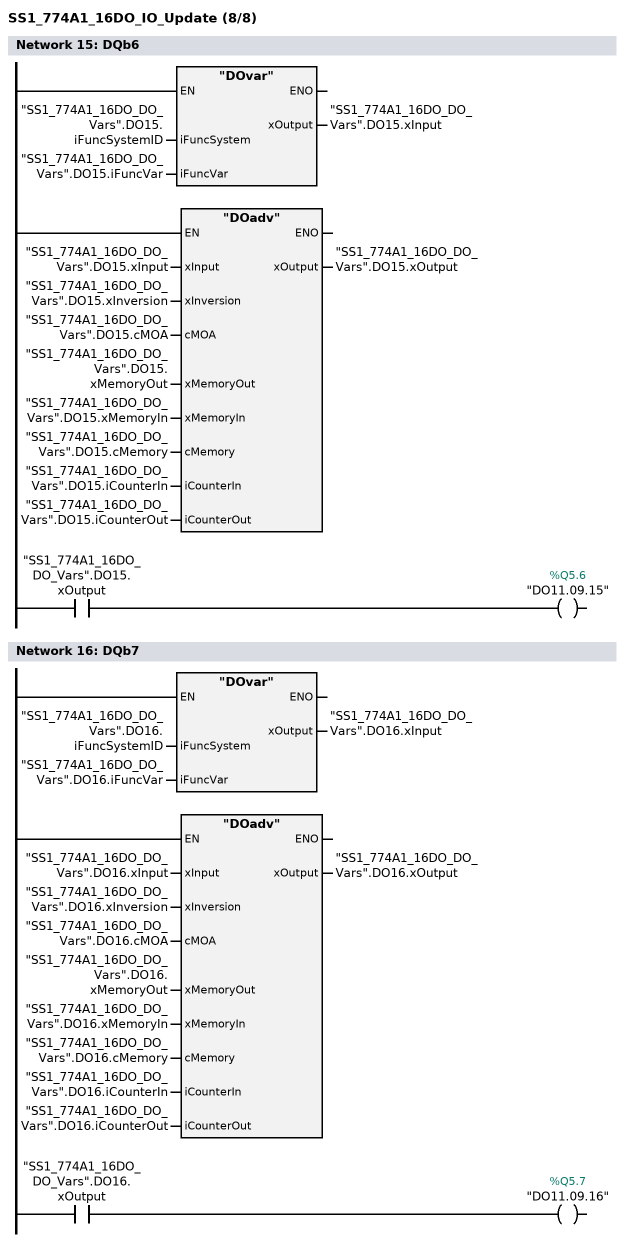
   RUNG wire#powerrail
      "DOvar"(iFuncSystem := "SS1_774A1_16DO_DO_Vars".DO15.iFuncSystemID, iFuncVar := "SS1_774A1_16DO_DO_Vars".DO15.iFuncVar, xOutput => "SS1_774A1_16DO_DO_Vars".DO15.xInput)
   END_RUNG
   RUNG wire#powerrail
      "DOadv"(xInput := "SS1_774A1_16DO_DO_Vars".DO15.xInput, xInversion := "SS1_774A1_16DO_DO_Vars".DO15.xInversion, cMOA := "SS1_774A1_16DO_DO_Vars".DO15.cMOA, xMemoryOut := "SS1_774A1_16DO_DO_Vars".DO15.xMemoryOut, xMemoryIn := "SS1_774A1_16DO_DO_Vars".DO15.xMemoryIn, cMemory := "SS1_774A1_16DO_DO_Vars".DO15.cMemory, iCounterIn := "SS1_774A1_16DO_DO_Vars".DO15.iCounterIn, iCounterOut := "SS1_774A1_16DO_DO_Vars".DO15.iCounterOut, xOutput => "SS1_774A1_16DO_DO_Vars".DO15.xOutput)
   END_RUNG
   RUNG wire#powerrail
      Contact( "SS1_774A1_16DO_DO_Vars".DO15.xOutput )
      Coil( "DO11.09.15" )
   END_RUNG
   // the same network as SCL:
   "DOvar"(iFuncSystem := "SS1_774A1_16DO_DO_Vars".DO15.iFuncSystemID,
           iFuncVar := "SS1_774A1_16DO_DO_Vars".DO15.iFuncVar,
           xOutput => "SS1_774A1_16DO_DO_Vars".DO15.xInput);
   "DOadv"(xInput := "SS1_774A1_16DO_DO_Vars".DO15.xInput,
           xInversion := "SS1_774A1_16DO_DO_Vars".DO15.xInversion,
           cMOA := "SS1_774A1_16DO_DO_Vars".DO15.cMOA,
           xMemoryOut := "SS1_774A1_16DO_DO_Vars".DO15.xMemoryOut,
           xMemoryIn := "SS1_774A1_16DO_DO_Vars".DO15.xMemoryIn,
           cMemory := "SS1_774A1_16DO_DO_Vars".DO15.cMemory,
           iCounterIn := "SS1_774A1_16DO_DO_Vars".DO15.iCounterIn,
           iCounterOut := "SS1_774A1_16DO_DO_Vars".DO15.iCounterOut,
           xOutput => "SS1_774A1_16DO_DO_Vars".DO15.xOutput);
   "DO11.09.15" := "SS1_774A1_16DO_DO_Vars".DO15.xOutput;
END_REGION

REGION Network 16: DQb7
   RUNG wire#powerrail
      "DOvar"(iFuncSystem := "SS1_774A1_16DO_DO_Vars".DO16.iFuncSystemID, iFuncVar := "SS1_774A1_16DO_DO_Vars".DO16.iFuncVar, xOutput => "SS1_774A1_16DO_DO_Vars".DO16.xInput)
   END_RUNG
   RUNG wire#powerrail
      "DOadv"(xInput := "SS1_774A1_16DO_DO_Vars".DO16.xInput, xInversion := "SS1_774A1_16DO_DO_Vars".DO16.xInversion, cMOA := "SS1_774A1_16DO_DO_Vars".DO16.cMOA, xMemoryOut := "SS1_774A1_16DO_DO_Vars".DO16.xMemoryOut, xMemoryIn := "SS1_774A1_16DO_DO_Vars".DO16.xMemoryIn, cMemory := "SS1_774A1_16DO_DO_Vars".DO16.cMemory, iCounterIn := "SS1_774A1_16DO_DO_Vars".DO16.iCounterIn, iCounterOut := "SS1_774A1_16DO_DO_Vars".DO16.iCounterOut, xOutput => "SS1_774A1_16DO_DO_Vars".DO16.xOutput)
   END_RUNG
   RUNG wire#powerrail
      Contact( "SS1_774A1_16DO_DO_Vars".DO16.xOutput )
      Coil( "DO11.09.16" )
   END_RUNG
   // the same network as SCL:
   "DOvar"(iFuncSystem := "SS1_774A1_16DO_DO_Vars".DO16.iFuncSystemID,
           iFuncVar := "SS1_774A1_16DO_DO_Vars".DO16.iFuncVar,
           xOutput => "SS1_774A1_16DO_DO_Vars".DO16.xInput);
   "DOadv"(xInput := "SS1_774A1_16DO_DO_Vars".DO16.xInput,
           xInversion := "SS1_774A1_16DO_DO_Vars".DO16.xInversion,
           cMOA := "SS1_774A1_16DO_DO_Vars".DO16.cMOA,
           xMemoryOut := "SS1_774A1_16DO_DO_Vars".DO16.xMemoryOut,
           xMemoryIn := "SS1_774A1_16DO_DO_Vars".DO16.xMemoryIn,
           cMemory := "SS1_774A1_16DO_DO_Vars".DO16.cMemory,
           iCounterIn := "SS1_774A1_16DO_DO_Vars".DO16.iCounterIn,
           iCounterOut := "SS1_774A1_16DO_DO_Vars".DO16.iCounterOut,
           xOutput => "SS1_774A1_16DO_DO_Vars".DO16.xOutput);
   "DO11.09.16" := "SS1_774A1_16DO_DO_Vars".DO16.xOutput;
END_REGION
END_FUNCTION

FUNCTION "SS1_780A1_8AI_IO_Update" : Void   // FC11030, LAD
{ S7_Optimized_Access := 'TRUE' }
VERSION : 0.1
// stored: AutoNumber false, IsIECCheckEnabled false, SetENOAutomatically false, UDAEnableTagReadback false
BEGIN

REGION Network 1: AI0
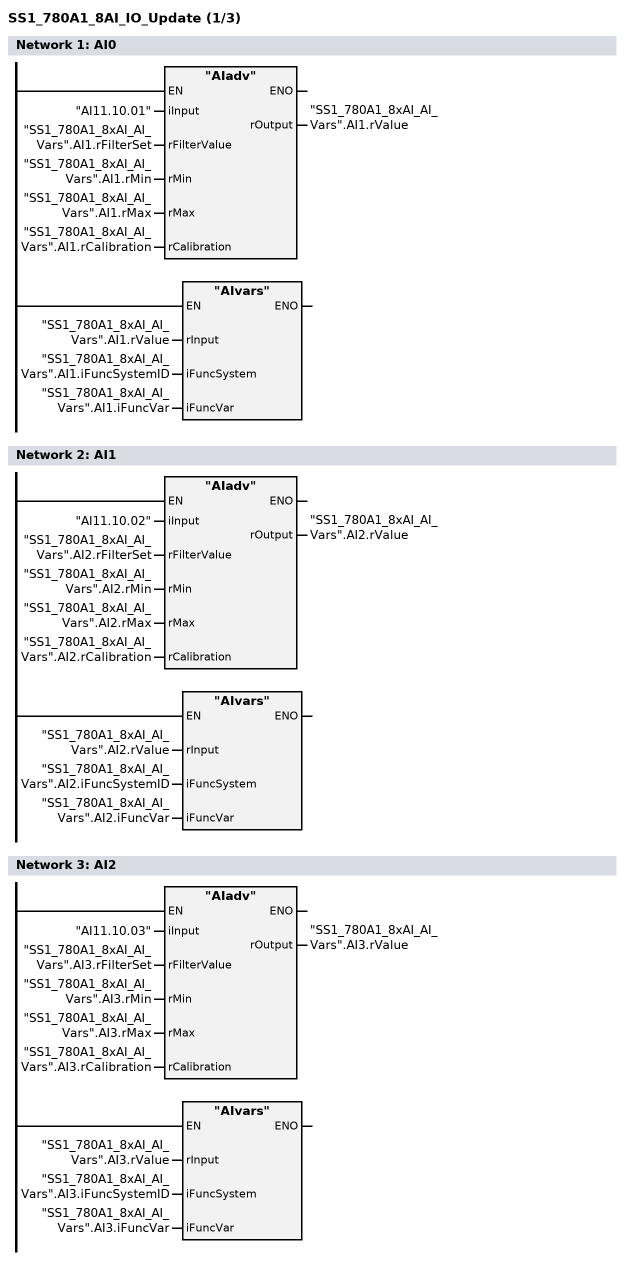
   RUNG wire#powerrail
      "AIadv"(iInput := "AI11.10.01", rFilterValue := "SS1_780A1_8xAI_AI_Vars".AI1.rFilterSet, rMin := "SS1_780A1_8xAI_AI_Vars".AI1.rMin, rMax := "SS1_780A1_8xAI_AI_Vars".AI1.rMax, rCalibration := "SS1_780A1_8xAI_AI_Vars".AI1.rCalibration, rOutput => "SS1_780A1_8xAI_AI_Vars".AI1.rValue)
   END_RUNG
   RUNG wire#powerrail
      "AIvars"(rInput := "SS1_780A1_8xAI_AI_Vars".AI1.rValue, iFuncSystem := "SS1_780A1_8xAI_AI_Vars".AI1.iFuncSystemID, iFuncVar := "SS1_780A1_8xAI_AI_Vars".AI1.iFuncVar)
   END_RUNG
   // the same network as SCL:
   "AIadv"(iInput := "AI11.10.01",
           rFilterValue := "SS1_780A1_8xAI_AI_Vars".AI1.rFilterSet,
           rMin := "SS1_780A1_8xAI_AI_Vars".AI1.rMin,
           rMax := "SS1_780A1_8xAI_AI_Vars".AI1.rMax,
           rCalibration := "SS1_780A1_8xAI_AI_Vars".AI1.rCalibration,
           rOutput => "SS1_780A1_8xAI_AI_Vars".AI1.rValue);
   "AIvars"(rInput := "SS1_780A1_8xAI_AI_Vars".AI1.rValue,
            iFuncSystem := "SS1_780A1_8xAI_AI_Vars".AI1.iFuncSystemID,
            iFuncVar := "SS1_780A1_8xAI_AI_Vars".AI1.iFuncVar);
END_REGION

REGION Network 2: AI1
   RUNG wire#powerrail
      "AIadv"(iInput := "AI11.10.02", rFilterValue := "SS1_780A1_8xAI_AI_Vars".AI2.rFilterSet, rMin := "SS1_780A1_8xAI_AI_Vars".AI2.rMin, rMax := "SS1_780A1_8xAI_AI_Vars".AI2.rMax, rCalibration := "SS1_780A1_8xAI_AI_Vars".AI2.rCalibration, rOutput => "SS1_780A1_8xAI_AI_Vars".AI2.rValue)
   END_RUNG
   RUNG wire#powerrail
      "AIvars"(rInput := "SS1_780A1_8xAI_AI_Vars".AI2.rValue, iFuncSystem := "SS1_780A1_8xAI_AI_Vars".AI2.iFuncSystemID, iFuncVar := "SS1_780A1_8xAI_AI_Vars".AI2.iFuncVar)
   END_RUNG
   // the same network as SCL:
   "AIadv"(iInput := "AI11.10.02",
           rFilterValue := "SS1_780A1_8xAI_AI_Vars".AI2.rFilterSet,
           rMin := "SS1_780A1_8xAI_AI_Vars".AI2.rMin,
           rMax := "SS1_780A1_8xAI_AI_Vars".AI2.rMax,
           rCalibration := "SS1_780A1_8xAI_AI_Vars".AI2.rCalibration,
           rOutput => "SS1_780A1_8xAI_AI_Vars".AI2.rValue);
   "AIvars"(rInput := "SS1_780A1_8xAI_AI_Vars".AI2.rValue,
            iFuncSystem := "SS1_780A1_8xAI_AI_Vars".AI2.iFuncSystemID,
            iFuncVar := "SS1_780A1_8xAI_AI_Vars".AI2.iFuncVar);
END_REGION

REGION Network 3: AI2
   RUNG wire#powerrail
      "AIadv"(iInput := "AI11.10.03", rFilterValue := "SS1_780A1_8xAI_AI_Vars".AI3.rFilterSet, rMin := "SS1_780A1_8xAI_AI_Vars".AI3.rMin, rMax := "SS1_780A1_8xAI_AI_Vars".AI3.rMax, rCalibration := "SS1_780A1_8xAI_AI_Vars".AI3.rCalibration, rOutput => "SS1_780A1_8xAI_AI_Vars".AI3.rValue)
   END_RUNG
   RUNG wire#powerrail
      "AIvars"(rInput := "SS1_780A1_8xAI_AI_Vars".AI3.rValue, iFuncSystem := "SS1_780A1_8xAI_AI_Vars".AI3.iFuncSystemID, iFuncVar := "SS1_780A1_8xAI_AI_Vars".AI3.iFuncVar)
   END_RUNG
   // the same network as SCL:
   "AIadv"(iInput := "AI11.10.03",
           rFilterValue := "SS1_780A1_8xAI_AI_Vars".AI3.rFilterSet,
           rMin := "SS1_780A1_8xAI_AI_Vars".AI3.rMin,
           rMax := "SS1_780A1_8xAI_AI_Vars".AI3.rMax,
           rCalibration := "SS1_780A1_8xAI_AI_Vars".AI3.rCalibration,
           rOutput => "SS1_780A1_8xAI_AI_Vars".AI3.rValue);
   "AIvars"(rInput := "SS1_780A1_8xAI_AI_Vars".AI3.rValue,
            iFuncSystem := "SS1_780A1_8xAI_AI_Vars".AI3.iFuncSystemID,
            iFuncVar := "SS1_780A1_8xAI_AI_Vars".AI3.iFuncVar);
END_REGION

REGION Network 4: AI3
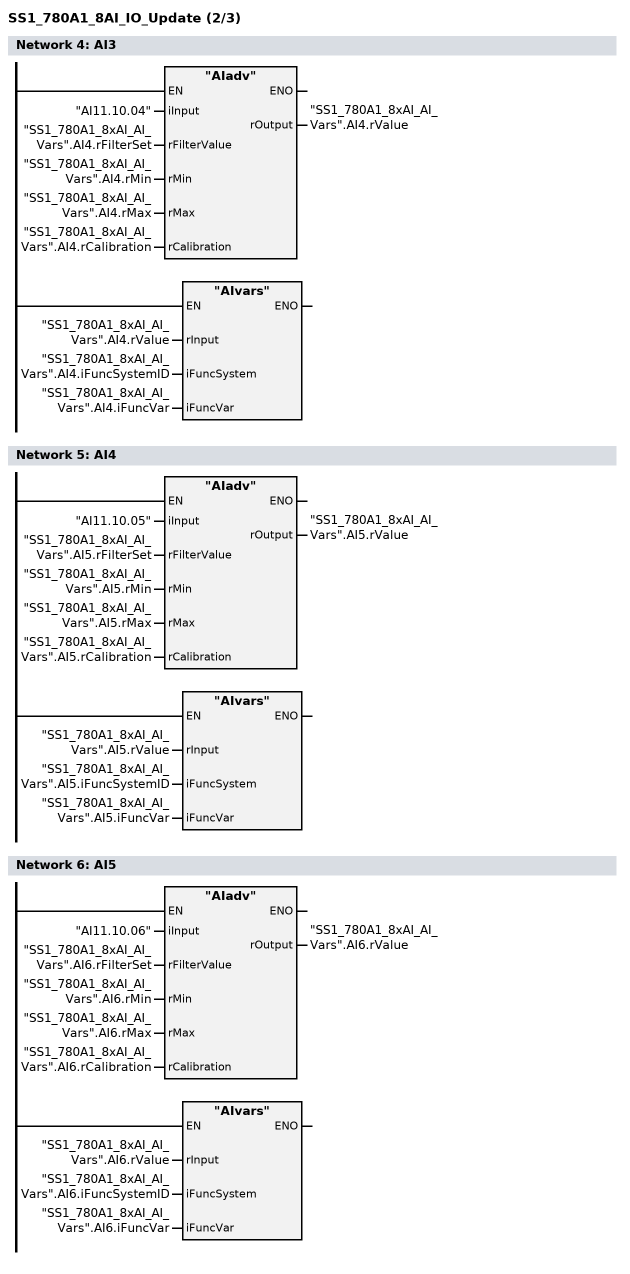
   RUNG wire#powerrail
      "AIadv"(iInput := "AI11.10.04", rFilterValue := "SS1_780A1_8xAI_AI_Vars".AI4.rFilterSet, rMin := "SS1_780A1_8xAI_AI_Vars".AI4.rMin, rMax := "SS1_780A1_8xAI_AI_Vars".AI4.rMax, rCalibration := "SS1_780A1_8xAI_AI_Vars".AI4.rCalibration, rOutput => "SS1_780A1_8xAI_AI_Vars".AI4.rValue)
   END_RUNG
   RUNG wire#powerrail
      "AIvars"(rInput := "SS1_780A1_8xAI_AI_Vars".AI4.rValue, iFuncSystem := "SS1_780A1_8xAI_AI_Vars".AI4.iFuncSystemID, iFuncVar := "SS1_780A1_8xAI_AI_Vars".AI4.iFuncVar)
   END_RUNG
   // the same network as SCL:
   "AIadv"(iInput := "AI11.10.04",
           rFilterValue := "SS1_780A1_8xAI_AI_Vars".AI4.rFilterSet,
           rMin := "SS1_780A1_8xAI_AI_Vars".AI4.rMin,
           rMax := "SS1_780A1_8xAI_AI_Vars".AI4.rMax,
           rCalibration := "SS1_780A1_8xAI_AI_Vars".AI4.rCalibration,
           rOutput => "SS1_780A1_8xAI_AI_Vars".AI4.rValue);
   "AIvars"(rInput := "SS1_780A1_8xAI_AI_Vars".AI4.rValue,
            iFuncSystem := "SS1_780A1_8xAI_AI_Vars".AI4.iFuncSystemID,
            iFuncVar := "SS1_780A1_8xAI_AI_Vars".AI4.iFuncVar);
END_REGION

REGION Network 5: AI4
   RUNG wire#powerrail
      "AIadv"(iInput := "AI11.10.05", rFilterValue := "SS1_780A1_8xAI_AI_Vars".AI5.rFilterSet, rMin := "SS1_780A1_8xAI_AI_Vars".AI5.rMin, rMax := "SS1_780A1_8xAI_AI_Vars".AI5.rMax, rCalibration := "SS1_780A1_8xAI_AI_Vars".AI5.rCalibration, rOutput => "SS1_780A1_8xAI_AI_Vars".AI5.rValue)
   END_RUNG
   RUNG wire#powerrail
      "AIvars"(rInput := "SS1_780A1_8xAI_AI_Vars".AI5.rValue, iFuncSystem := "SS1_780A1_8xAI_AI_Vars".AI5.iFuncSystemID, iFuncVar := "SS1_780A1_8xAI_AI_Vars".AI5.iFuncVar)
   END_RUNG
   // the same network as SCL:
   "AIadv"(iInput := "AI11.10.05",
           rFilterValue := "SS1_780A1_8xAI_AI_Vars".AI5.rFilterSet,
           rMin := "SS1_780A1_8xAI_AI_Vars".AI5.rMin,
           rMax := "SS1_780A1_8xAI_AI_Vars".AI5.rMax,
           rCalibration := "SS1_780A1_8xAI_AI_Vars".AI5.rCalibration,
           rOutput => "SS1_780A1_8xAI_AI_Vars".AI5.rValue);
   "AIvars"(rInput := "SS1_780A1_8xAI_AI_Vars".AI5.rValue,
            iFuncSystem := "SS1_780A1_8xAI_AI_Vars".AI5.iFuncSystemID,
            iFuncVar := "SS1_780A1_8xAI_AI_Vars".AI5.iFuncVar);
END_REGION

REGION Network 6: AI5
   RUNG wire#powerrail
      "AIadv"(iInput := "AI11.10.06", rFilterValue := "SS1_780A1_8xAI_AI_Vars".AI6.rFilterSet, rMin := "SS1_780A1_8xAI_AI_Vars".AI6.rMin, rMax := "SS1_780A1_8xAI_AI_Vars".AI6.rMax, rCalibration := "SS1_780A1_8xAI_AI_Vars".AI6.rCalibration, rOutput => "SS1_780A1_8xAI_AI_Vars".AI6.rValue)
   END_RUNG
   RUNG wire#powerrail
      "AIvars"(rInput := "SS1_780A1_8xAI_AI_Vars".AI6.rValue, iFuncSystem := "SS1_780A1_8xAI_AI_Vars".AI6.iFuncSystemID, iFuncVar := "SS1_780A1_8xAI_AI_Vars".AI6.iFuncVar)
   END_RUNG
   // the same network as SCL:
   "AIadv"(iInput := "AI11.10.06",
           rFilterValue := "SS1_780A1_8xAI_AI_Vars".AI6.rFilterSet,
           rMin := "SS1_780A1_8xAI_AI_Vars".AI6.rMin,
           rMax := "SS1_780A1_8xAI_AI_Vars".AI6.rMax,
           rCalibration := "SS1_780A1_8xAI_AI_Vars".AI6.rCalibration,
           rOutput => "SS1_780A1_8xAI_AI_Vars".AI6.rValue);
   "AIvars"(rInput := "SS1_780A1_8xAI_AI_Vars".AI6.rValue,
            iFuncSystem := "SS1_780A1_8xAI_AI_Vars".AI6.iFuncSystemID,
            iFuncVar := "SS1_780A1_8xAI_AI_Vars".AI6.iFuncVar);
END_REGION

REGION Network 7: AI6
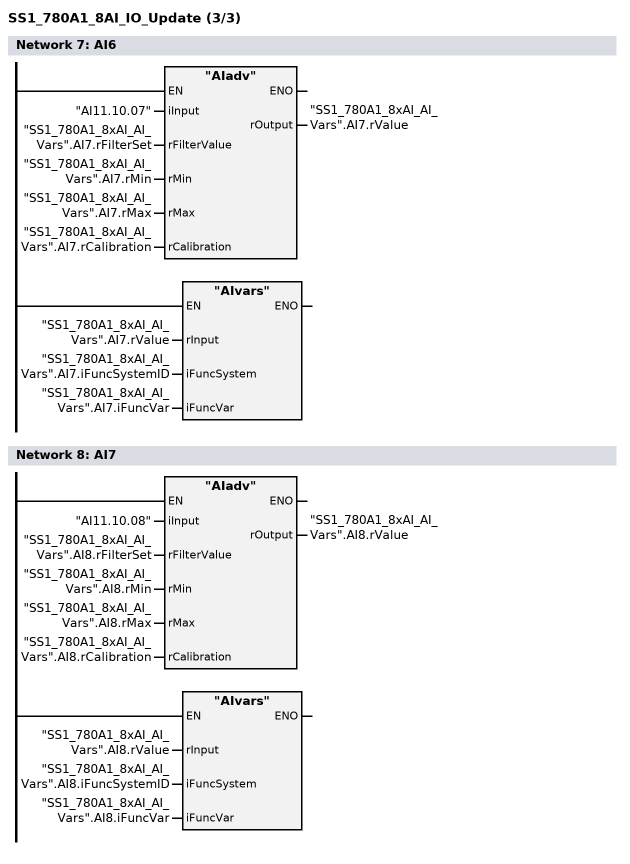
   RUNG wire#powerrail
      "AIadv"(iInput := "AI11.10.07", rFilterValue := "SS1_780A1_8xAI_AI_Vars".AI7.rFilterSet, rMin := "SS1_780A1_8xAI_AI_Vars".AI7.rMin, rMax := "SS1_780A1_8xAI_AI_Vars".AI7.rMax, rCalibration := "SS1_780A1_8xAI_AI_Vars".AI7.rCalibration, rOutput => "SS1_780A1_8xAI_AI_Vars".AI7.rValue)
   END_RUNG
   RUNG wire#powerrail
      "AIvars"(rInput := "SS1_780A1_8xAI_AI_Vars".AI7.rValue, iFuncSystem := "SS1_780A1_8xAI_AI_Vars".AI7.iFuncSystemID, iFuncVar := "SS1_780A1_8xAI_AI_Vars".AI7.iFuncVar)
   END_RUNG
   // the same network as SCL:
   "AIadv"(iInput := "AI11.10.07",
           rFilterValue := "SS1_780A1_8xAI_AI_Vars".AI7.rFilterSet,
           rMin := "SS1_780A1_8xAI_AI_Vars".AI7.rMin,
           rMax := "SS1_780A1_8xAI_AI_Vars".AI7.rMax,
           rCalibration := "SS1_780A1_8xAI_AI_Vars".AI7.rCalibration,
           rOutput => "SS1_780A1_8xAI_AI_Vars".AI7.rValue);
   "AIvars"(rInput := "SS1_780A1_8xAI_AI_Vars".AI7.rValue,
            iFuncSystem := "SS1_780A1_8xAI_AI_Vars".AI7.iFuncSystemID,
            iFuncVar := "SS1_780A1_8xAI_AI_Vars".AI7.iFuncVar);
END_REGION

REGION Network 8: AI7
   RUNG wire#powerrail
      "AIadv"(iInput := "AI11.10.08", rFilterValue := "SS1_780A1_8xAI_AI_Vars".AI8.rFilterSet, rMin := "SS1_780A1_8xAI_AI_Vars".AI8.rMin, rMax := "SS1_780A1_8xAI_AI_Vars".AI8.rMax, rCalibration := "SS1_780A1_8xAI_AI_Vars".AI8.rCalibration, rOutput => "SS1_780A1_8xAI_AI_Vars".AI8.rValue)
   END_RUNG
   RUNG wire#powerrail
      "AIvars"(rInput := "SS1_780A1_8xAI_AI_Vars".AI8.rValue, iFuncSystem := "SS1_780A1_8xAI_AI_Vars".AI8.iFuncSystemID, iFuncVar := "SS1_780A1_8xAI_AI_Vars".AI8.iFuncVar)
   END_RUNG
   // the same network as SCL:
   "AIadv"(iInput := "AI11.10.08",
           rFilterValue := "SS1_780A1_8xAI_AI_Vars".AI8.rFilterSet,
           rMin := "SS1_780A1_8xAI_AI_Vars".AI8.rMin,
           rMax := "SS1_780A1_8xAI_AI_Vars".AI8.rMax,
           rCalibration := "SS1_780A1_8xAI_AI_Vars".AI8.rCalibration,
           rOutput => "SS1_780A1_8xAI_AI_Vars".AI8.rValue);
   "AIvars"(rInput := "SS1_780A1_8xAI_AI_Vars".AI8.rValue,
            iFuncSystem := "SS1_780A1_8xAI_AI_Vars".AI8.iFuncSystemID,
            iFuncVar := "SS1_780A1_8xAI_AI_Vars".AI8.iFuncVar);
END_REGION
END_FUNCTION

FUNCTION "SS1_784A1_4AO_IO_Update" : Void   // FC11040, LAD
{ S7_Optimized_Access := 'TRUE' }
VERSION : 0.1
// stored: AutoNumber false, IsIECCheckEnabled false, SetENOAutomatically false, UDAEnableTagReadback false
BEGIN

REGION Network 1: AO0
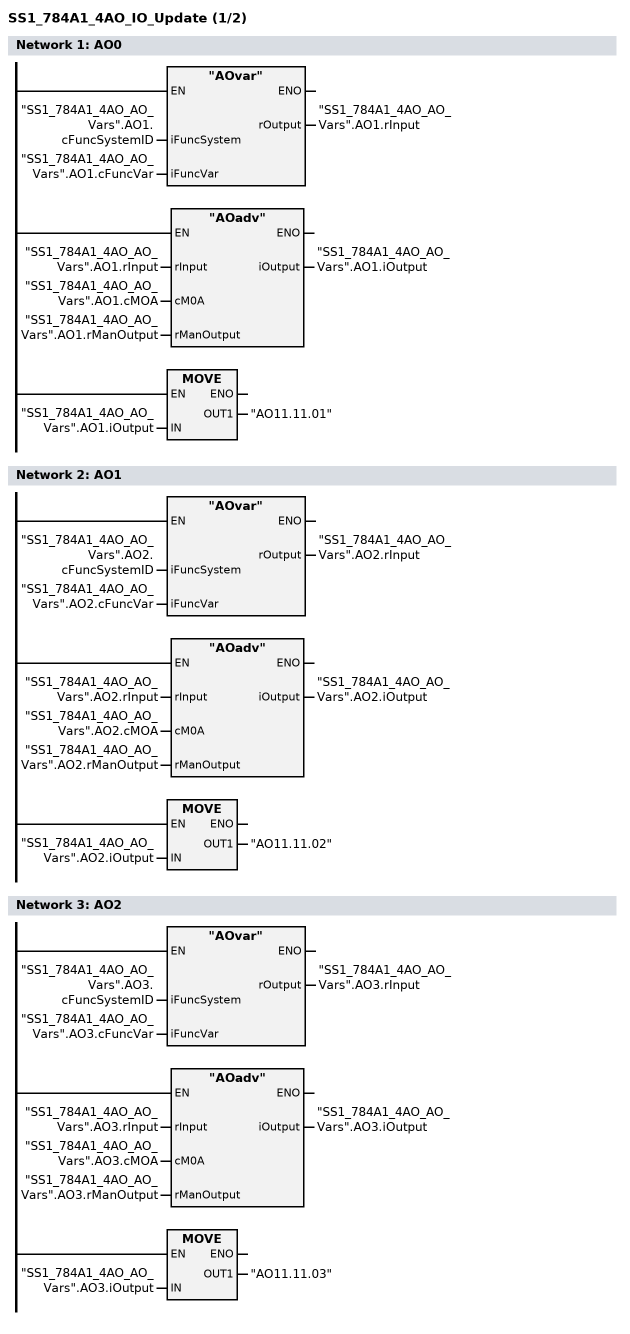
   RUNG wire#powerrail
      "AOvar"(iFuncSystem := "SS1_784A1_4AO_AO_Vars".AO1.cFuncSystemID, iFuncVar := "SS1_784A1_4AO_AO_Vars".AO1.cFuncVar, rOutput => "SS1_784A1_4AO_AO_Vars".AO1.rInput)
   END_RUNG
   RUNG wire#powerrail
      "AOadv"(rInput := "SS1_784A1_4AO_AO_Vars".AO1.rInput, cM0A := "SS1_784A1_4AO_AO_Vars".AO1.cMOA, rManOutput := "SS1_784A1_4AO_AO_Vars".AO1.rManOutput, iOutput => "SS1_784A1_4AO_AO_Vars".AO1.iOutput)
   END_RUNG
   RUNG wire#powerrail
      Move(in := "SS1_784A1_4AO_AO_Vars".AO1.iOutput, out1 => "AO11.11.01")
   END_RUNG
   // the same network as SCL:
   "AOvar"(iFuncSystem := "SS1_784A1_4AO_AO_Vars".AO1.cFuncSystemID,
           iFuncVar := "SS1_784A1_4AO_AO_Vars".AO1.cFuncVar,
           rOutput => "SS1_784A1_4AO_AO_Vars".AO1.rInput);
   "AOadv"(rInput := "SS1_784A1_4AO_AO_Vars".AO1.rInput,
           cM0A := "SS1_784A1_4AO_AO_Vars".AO1.cMOA,
           rManOutput := "SS1_784A1_4AO_AO_Vars".AO1.rManOutput,
           iOutput => "SS1_784A1_4AO_AO_Vars".AO1.iOutput);
   "AO11.11.01" := "SS1_784A1_4AO_AO_Vars".AO1.iOutput;
END_REGION

REGION Network 2: AO1
   RUNG wire#powerrail
      "AOvar"(iFuncSystem := "SS1_784A1_4AO_AO_Vars".AO2.cFuncSystemID, iFuncVar := "SS1_784A1_4AO_AO_Vars".AO2.cFuncVar, rOutput => "SS1_784A1_4AO_AO_Vars".AO2.rInput)
   END_RUNG
   RUNG wire#powerrail
      "AOadv"(rInput := "SS1_784A1_4AO_AO_Vars".AO2.rInput, cM0A := "SS1_784A1_4AO_AO_Vars".AO2.cMOA, rManOutput := "SS1_784A1_4AO_AO_Vars".AO2.rManOutput, iOutput => "SS1_784A1_4AO_AO_Vars".AO2.iOutput)
   END_RUNG
   RUNG wire#powerrail
      Move(in := "SS1_784A1_4AO_AO_Vars".AO2.iOutput, out1 => "AO11.11.02")
   END_RUNG
   // the same network as SCL:
   "AOvar"(iFuncSystem := "SS1_784A1_4AO_AO_Vars".AO2.cFuncSystemID,
           iFuncVar := "SS1_784A1_4AO_AO_Vars".AO2.cFuncVar,
           rOutput => "SS1_784A1_4AO_AO_Vars".AO2.rInput);
   "AOadv"(rInput := "SS1_784A1_4AO_AO_Vars".AO2.rInput,
           cM0A := "SS1_784A1_4AO_AO_Vars".AO2.cMOA,
           rManOutput := "SS1_784A1_4AO_AO_Vars".AO2.rManOutput,
           iOutput => "SS1_784A1_4AO_AO_Vars".AO2.iOutput);
   "AO11.11.02" := "SS1_784A1_4AO_AO_Vars".AO2.iOutput;
END_REGION

REGION Network 3: AO2
   RUNG wire#powerrail
      "AOvar"(iFuncSystem := "SS1_784A1_4AO_AO_Vars".AO3.cFuncSystemID, iFuncVar := "SS1_784A1_4AO_AO_Vars".AO3.cFuncVar, rOutput => "SS1_784A1_4AO_AO_Vars".AO3.rInput)
   END_RUNG
   RUNG wire#powerrail
      "AOadv"(rInput := "SS1_784A1_4AO_AO_Vars".AO3.rInput, cM0A := "SS1_784A1_4AO_AO_Vars".AO3.cMOA, rManOutput := "SS1_784A1_4AO_AO_Vars".AO3.rManOutput, iOutput => "SS1_784A1_4AO_AO_Vars".AO3.iOutput)
   END_RUNG
   RUNG wire#powerrail
      Move(in := "SS1_784A1_4AO_AO_Vars".AO3.iOutput, out1 => "AO11.11.03")
   END_RUNG
   // the same network as SCL:
   "AOvar"(iFuncSystem := "SS1_784A1_4AO_AO_Vars".AO3.cFuncSystemID,
           iFuncVar := "SS1_784A1_4AO_AO_Vars".AO3.cFuncVar,
           rOutput => "SS1_784A1_4AO_AO_Vars".AO3.rInput);
   "AOadv"(rInput := "SS1_784A1_4AO_AO_Vars".AO3.rInput,
           cM0A := "SS1_784A1_4AO_AO_Vars".AO3.cMOA,
           rManOutput := "SS1_784A1_4AO_AO_Vars".AO3.rManOutput,
           iOutput => "SS1_784A1_4AO_AO_Vars".AO3.iOutput);
   "AO11.11.03" := "SS1_784A1_4AO_AO_Vars".AO3.iOutput;
END_REGION

REGION Network 4: AO3
